    |   movel([0.251673, -1.221759, -2.667128, -0.823502, 1.570796, 1.822469],accel_mss,speed_ms,0,blend_radius_m)
    |   movel([0.252256, -1.224586, -2.665710, -0.822093, 1.570796, 1.823052],accel_mss,speed_ms,0,blend_radius_m)
    |   movel([0.252313, -1.225370, -2.665315, -0.821704, 1.570796, 1.823110],accel_mss,speed_ms,0,blend_radius_m)
    |   movel([0.252119, -1.226392, -2.664799, -0.821198, 1.570796, 1.822915],accel_mss,speed_ms,0,blend_radius_m)
    |   movel([0.252114, -1.226648, -2.664669, -0.821071, 1.570796, 1.822911],accel_mss,speed_ms,0,blend_radius_m)
    |   movel([0.252664, -1.227115, -2.664433, -0.820840, 1.570796, 1.823460],accel_mss,speed_ms,0,blend_radius_m)
    |   movel([0.252892, -1.227914, -2.664028, -0.820447, 1.570796, 1.823688],accel_mss,speed_ms,0,blend_radius_m)
    |   movel([0.253520, -1.231694, -2.662103, -0.818592, 1.570796, 1.824316],accel_mss,speed_ms,0,blend_radius_m)
    |   movel([0.254096, -1.235374, -2.660213, -0.816803, 1.570796, 1.824892],accel_mss,speed_ms,0,blend_radius_m)
    |   movel([0.255273, -1.240979, -2.657303, -0.814107, 1.570796, 1.826070],accel_mss,speed_ms,0,blend_radius_m)
    |   movel([0.255921, -1.243115, -2.656184, -0.813089, 1.570796, 1.826717],accel_mss,speed_ms,0,blend_radius_m)
    |   movel([0.256893, -1.245588, -2.654883, -0.811918, 1.570796, 1.827689],accel_mss,speed_ms,0,blend_radius_m)
    |   movel([0.258056, -1.247911, -2.653653, -0.810825, 1.570796, 1.828852],accel_mss,speed_ms,0,blend_radius_m)
    |   movel([0.259299, -1.249832, -2.652632, -0.809925, 1.570796, 1.830095],accel_mss,speed_ms,0,blend_radius_m)
    |   movel([0.260770, -1.251552, -2.651713, -0.809124, 1.570796, 1.831566],accel_mss,speed_ms,0,blend_radius_m)
    |   movel([0.262149, -1.252766, -2.651063, -0.808560, 1.570796, 1.832945],accel_mss,speed_ms,0,blend_radius_m)
    |   movel([0.263720, -1.253774, -2.650522, -0.808094, 1.570796, 1.834516],accel_mss,speed_ms,0,blend_radius_m)
    |   movel([0.265017, -1.254154, -2.650317, -0.807918, 1.570796, 1.835813],accel_mss,speed_ms,0,blend_radius_m)
    |   movel([0.266576, -1.254061, -2.650367, -0.807961, 1.570796, 1.837372],accel_mss,speed_ms,0,blend_radius_m)
    |   movel([0.268162, -1.253521, -2.650657, -0.808210, 1.570796, 1.838958],accel_mss,speed_ms,0,blend_radius_m)
    |   movel([0.268641, -1.253267, -2.650794, -0.808328, 1.570796, 1.839437],accel_mss,speed_ms,0,blend_radius_m)
    |   movel([0.270173, -1.252133, -2.651402, -0.808854, 1.570796, 1.840969],accel_mss,speed_ms,0,blend_radius_m)
    |   movel([0.271779, -1.250504, -2.652273, -0.809612, 1.570796, 1.842575],accel_mss,speed_ms,0,blend_radius_m)
    |   movel([0.273303, -1.248559, -2.653309, -0.810521, 1.570796, 1.844100],accel_mss,speed_ms,0,blend_radius_m)
    |   movel([0.274592, -1.246469, -2.654417, -0.811503, 1.570796, 1.845389],accel_mss,speed_ms,0,blend_radius_m)
    |   movel([0.275448, -1.244543, -2.655434, -0.812412, 1.570796, 1.846245],accel_mss,speed_ms,0,blend_radius_m)
    |   movel([0.276254, -1.241932, -2.656805, -0.813652, 1.570796, 1.847050],accel_mss,speed_ms,0,blend_radius_m)
    |   movel([0.276891, -1.239150, -2.658257, -0.814983, 1.570796, 1.847687],accel_mss,speed_ms,0,blend_radius_m)
    |   movel([0.277227, -1.236646, -2.659556, -0.816187, 1.570796, 1.848023],accel_mss,speed_ms,0,blend_radius_m)
    |   movel([0.277345, -1.234191, -2.660822, -0.817376, 1.570796, 1.848141],accel_mss,speed_ms,0,blend_radius_m)
    |   movel([0.277297, -1.231803, -2.662047, -0.818539, 1.570796, 1.848093],accel_mss,speed_ms,0,blend_radius_m)
    |   movel([0.277086, -1.229560, -2.663192, -0.819637, 1.570796, 1.847882],accel_mss,speed_ms,0,blend_radius_m)
    |   movel([0.276698, -1.227409, -2.664285, -0.820696, 1.570796, 1.847494],accel_mss,speed_ms,0,blend_radius_m)
    |   movel([0.276147, -1.225413, -2.665293, -0.821683, 1.570796, 1.846943],accel_mss,speed_ms,0,blend_radius_m)
    |   movel([0.275424, -1.223525, -2.666243, -0.822621, 1.570796, 1.846220],accel_mss,speed_ms,0,blend_radius_m)
    |   movel([0.274540, -1.221803, -2.667106, -0.823480, 1.570796, 1.845336],accel_mss,speed_ms,0,blend_radius_m)
    |   movel([0.273482, -1.220215, -2.667899, -0.824275, 1.570796, 1.844278],accel_mss,speed_ms,0,blend_radius_m)
    |   movel([0.272482, -1.219065, -2.668471, -0.824852, 1.570796, 1.843279],accel_mss,speed_ms,0,blend_radius_m)
    |   movel([0.272133, -1.218838, -2.668584, -0.824967, 1.570796, 1.842930],accel_mss,speed_ms,0,blend_radius_m)
    |   movel([0.271831, -1.218816, -2.668595, -0.824978, 1.570796, 1.842627],accel_mss,speed_ms,0,blend_radius_m)
    |   movel([0.271376, -1.219063, -2.668473, -0.824854, 1.570796, 1.842172],accel_mss,speed_ms,0,blend_radius_m)
    |   movel([0.271187, -1.219431, -2.668289, -0.824668, 1.570796, 1.841984],accel_mss,speed_ms,0,blend_radius_m)
    |   movel([0.271361, -1.219988, -2.668012, -0.824389, 1.570796, 1.842158],accel_mss,speed_ms,0,blend_radius_m)
    |   movel([0.271964, -1.220817, -2.667599, -0.823973, 1.570796, 1.842761],accel_mss,speed_ms,0,blend_radius_m)
    |   movel([0.273182, -1.222548, -2.666734, -0.823108, 1.570796, 1.843978],accel_mss,speed_ms,0,blend_radius_m)
    |   movel([0.274184, -1.224447, -2.665780, -0.822162, 1.570796, 1.844980],accel_mss,speed_ms,0,blend_radius_m)
    |   movel([0.274992, -1.226530, -2.664729, -0.821130, 1.570796, 1.845788],accel_mss,speed_ms,0,blend_radius_m)
    |   movel([0.275580, -1.228751, -2.663604, -0.820035, 1.570796, 1.846376],accel_mss,speed_ms,0,blend_radius_m)
    |   movel([0.275960, -1.231114, -2.662400, -0.818876, 1.570796, 1.846756],accel_mss,speed_ms,0,blend_radius_m)
    |   movel([0.276124, -1.233583, -2.661135, -0.817671, 1.570796, 1.846920],accel_mss,speed_ms,0,blend_radius_m)
    |   movel([0.276071, -1.236144, -2.659815, -0.816430, 1.570796, 1.846867],accel_mss,speed_ms,0,blend_radius_m)
    |   movel([0.275805, -1.238781, -2.658448, -0.815159, 1.570796, 1.846602],accel_mss,speed_ms,0,blend_radius_m)
    |   movel([0.275419, -1.240897, -2.657346, -0.814146, 1.570796, 1.846215],accel_mss,speed_ms,0,blend_radius_m)
    |   movel([0.274837, -1.243056, -2.656215, -0.813117, 1.570796, 1.845633],accel_mss,speed_ms,0,blend_radius_m)
    |   movel([0.274120, -1.244995, -2.655195, -0.812198, 1.570796, 1.844916],accel_mss,speed_ms,0,blend_radius_m)
    |   movel([0.273176, -1.246938, -2.654169, -0.811282, 1.570796, 1.843972],accel_mss,speed_ms,0,blend_radius_m)
    |   movel([0.272189, -1.248540, -2.653319, -0.810530, 1.570796, 1.842985],accel_mss,speed_ms,0,blend_radius_m)
    |   movel([0.271011, -1.250081, -2.652499, -0.809809, 1.570796, 1.841807],accel_mss,speed_ms,0,blend_radius_m)
    |   movel([0.269852, -1.251241, -2.651879, -0.809268, 1.570796, 1.840649],accel_mss,speed_ms,0,blend_radius_m)
    |   movel([0.268535, -1.252186, -2.651374, -0.808829, 1.570796, 1.839332],accel_mss,speed_ms,0,blend_radius_m)
    |   movel([0.267582, -1.252648, -2.651126, -0.808615, 1.570796, 1.838378],accel_mss,speed_ms,0,blend_radius_m)
    |   movel([0.266683, -1.252879, -2.651002, -0.808507, 1.570796, 1.837480],accel_mss,speed_ms,0,blend_radius_m)
    |   movel([0.265766, -1.252881, -2.651001, -0.808507, 1.570796, 1.836563],accel_mss,speed_ms,0,blend_radius_m)
    |   movel([0.264751, -1.252662, -2.651119, -0.808608, 1.570796, 1.835547],accel_mss,speed_ms,0,blend_radius_m)
    |   movel([0.263859, -1.252274, -2.651327, -0.808788, 1.570796, 1.834655],accel_mss,speed_ms,0,blend_radius_m)
    |   movel([0.263122, -1.251705, -2.651631, -0.809052, 1.570796, 1.833919],accel_mss,speed_ms,0,blend_radius_m)
    |   movel([0.260735, -1.249084, -2.653030, -0.810275, 1.570796, 1.831531],accel_mss,speed_ms,0,blend_radius_m)
    |   movel([0.258421, -1.246199, -2.654560, -0.811630, 1.570796, 1.829217],accel_mss,speed_ms,0,blend_radius_m)
    |   movel([0.258350, -1.245788, -2.654777, -0.811824, 1.570796, 1.829146],accel_mss,speed_ms,0,blend_radius_m)
    |   movel([0.258596, -1.245287, -2.655042, -0.812060, 1.570796, 1.829392],accel_mss,speed_ms,0,blend_radius_m)
    |   movel([0.258596, -1.244631, -2.655387, -0.812370, 1.570796, 1.829393],accel_mss,speed_ms,0,blend_radius_m)
    |   movel([0.258518, -1.243848, -2.655800, -0.812742, 1.570796, 1.829314],accel_mss,speed_ms,0,blend_radius_m)
    |   movel([0.258893, -1.242963, -2.656264, -0.813162, 1.570796, 1.829689],accel_mss,speed_ms,0,blend_radius_m)
    |   movel([0.259695, -1.242085, -2.656725, -0.813579, 1.570796, 1.830491],accel_mss,speed_ms,0,blend_radius_m)
    |   movel([0.260821, -1.241329, -2.657120, -0.813940, 1.570796, 1.831618],accel_mss,speed_ms,0,blend_radius_m)
    |   movel([0.261962, -1.240850, -2.657371, -0.814169, 1.570796, 1.832758],accel_mss,speed_ms,0,blend_radius_m)
    |   movel([0.263259, -1.240549, -2.657527, -0.814312, 1.570796, 1.834056],accel_mss,speed_ms,0,blend_radius_m)
    |   movel([0.264431, -1.240462, -2.657573, -0.814354, 1.570796, 1.835227],accel_mss,speed_ms,0,blend_radius_m)
    |   movel([0.265143, -1.240658, -2.657471, -0.814260, 1.570796, 1.835939],accel_mss,speed_ms,0,blend_radius_m)
    |   movel([0.265362, -1.240773, -2.657411, -0.814205, 1.570796, 1.836158],accel_mss,speed_ms,0,blend_radius_m)
    |   movel([0.266050, -1.240887, -2.657351, -0.814151, 1.570796, 1.836847],accel_mss,speed_ms,0,blend_radius_m)
    |   movel([0.266350, -1.240866, -2.657362, -0.814161, 1.570796, 1.837146],accel_mss,speed_ms,0,blend_radius_m)
    |   movel([0.266402, -1.240980, -2.657303, -0.814107, 1.570796, 1.837198],accel_mss,speed_ms,0,blend_radius_m)
    |   movel([0.266237, -1.241186, -2.657195, -0.814008, 1.570796, 1.837033],accel_mss,speed_ms,0,blend_radius_m)
    |   movel([0.265247, -1.241887, -2.656828, -0.813674, 1.570796, 1.836043],accel_mss,speed_ms,0,blend_radius_m)
    |   movel([0.264579, -1.242566, -2.656473, -0.813351, 1.570796, 1.835376],accel_mss,speed_ms,0,blend_radius_m)
    |   movel([0.263427, -1.244142, -2.655645, -0.812602, 1.570796, 1.834224],accel_mss,speed_ms,0,blend_radius_m)
    |   movel([0.262984, -1.245097, -2.655142, -0.812150, 1.570796, 1.833780],accel_mss,speed_ms,0,blend_radius_m)
    |   movel([0.262406, -1.247398, -2.653925, -0.811066, 1.570796, 1.833203],accel_mss,speed_ms,0,blend_radius_m)
    |   movel([0.262377, -1.248322, -2.653435, -0.810632, 1.570796, 1.833173],accel_mss,speed_ms,0,blend_radius_m)
    |   movel([0.262798, -1.250016, -2.652534, -0.809839, 1.570796, 1.833595],accel_mss,speed_ms,0,blend_radius_m)
    |   movel([0.263763, -1.251456, -2.651764, -0.809168, 1.570796, 1.834559],accel_mss,speed_ms,0,blend_radius_m)
    |   movel([0.264797, -1.252084, -2.651429, -0.808877, 1.570796, 1.835593],accel_mss,speed_ms,0,blend_radius_m)
    |   movel([0.265194, -1.252000, -2.651474, -0.808915, 1.570796, 1.835990],accel_mss,speed_ms,0,blend_radius_m)
    |   movel([0.265517, -1.251643, -2.651665, -0.809082, 1.570796, 1.836314],accel_mss,speed_ms,0,blend_radius_m)
    |   movel([0.265537, -1.251456, -2.651764, -0.809168, 1.570796, 1.836334],accel_mss,speed_ms,0,blend_radius_m)
    |   movel([0.264819, -1.250247, -2.652411, -0.809732, 1.570796, 1.835616],accel_mss,speed_ms,0,blend_radius_m)
    |   movel([0.264102, -1.249179, -2.652979, -0.810230, 1.570796, 1.834899],accel_mss,speed_ms,0,blend_radius_m)
    |   movel([0.263717, -1.248165, -2.653518, -0.810705, 1.570796, 1.834513],accel_mss,speed_ms,0,blend_radius_m)
    |   movel([0.263635, -1.247105, -2.654081, -0.811204, 1.570796, 1.834431],accel_mss,speed_ms,0,blend_radius_m)
    |   movel([0.263836, -1.245902, -2.654717, -0.811770, 1.570796, 1.834632],accel_mss,speed_ms,0,blend_radius_m)
    |   movel([0.264366, -1.244503, -2.655455, -0.812431, 1.570796, 1.835162],accel_mss,speed_ms,0,blend_radius_m)
    |   movel([0.265141, -1.243328, -2.656073, -0.812988, 1.570796, 1.835937],accel_mss,speed_ms,0,blend_radius_m)
    |   movel([0.266125, -1.242431, -2.656543, -0.813414, 1.570796, 1.836921],accel_mss,speed_ms,0,blend_radius_m)
    |   movel([0.267647, -1.241694, -2.656929, -0.813766, 1.570796, 1.838444],accel_mss,speed_ms,0,blend_radius_m)
    |   movel([0.268011, -1.241513, -2.657024, -0.813852, 1.570796, 1.838807],accel_mss,speed_ms,0,blend_radius_m)
    |   movel([0.268485, -1.241158, -2.657209, -0.814021, 1.570796, 1.839281],accel_mss,speed_ms,0,blend_radius_m)
    |   movel([0.268713, -1.241026, -2.657278, -0.814084, 1.570796, 1.839509],accel_mss,speed_ms,0,blend_radius_m)
    |   movel([0.268748, -1.241410, -2.657078, -0.813901, 1.570796, 1.839544],accel_mss,speed_ms,0,blend_radius_m)
    |   movel([0.269472, -1.242542, -2.656485, -0.813362, 1.570796, 1.840268],accel_mss,speed_ms,0,blend_radius_m)
    |   movel([0.270218, -1.243593, -2.655933, -0.812862, 1.570796, 1.841015],accel_mss,speed_ms,0,blend_radius_m)
    |   movel([0.270715, -1.244043, -2.655697, -0.812649, 1.570796, 1.841511],accel_mss,speed_ms,0,blend_radius_m)
    |   movel([0.271107, -1.244195, -2.655617, -0.812577, 1.570796, 1.841903],accel_mss,speed_ms,0,blend_radius_m)
    |   movel([0.271501, -1.244167, -2.655632, -0.812590, 1.570796, 1.842297],accel_mss,speed_ms,0,blend_radius_m)
    |   movel([0.271816, -1.243974, -2.655733, -0.812682, 1.570796, 1.842613],accel_mss,speed_ms,0,blend_radius_m)
    |   movel([0.272009, -1.243666, -2.655895, -0.812828, 1.570796, 1.842805],accel_mss,speed_ms,0,blend_radius_m)
    |   movel([0.272002, -1.243499, -2.655983, -0.812907, 1.570796, 1.842799],accel_mss,speed_ms,0,blend_radius_m)
    |   movel([0.270423, -1.241210, -2.657183, -0.813997, 1.570796, 1.841220],accel_mss,speed_ms,0,blend_radius_m)
    |   movel([0.269852, -1.240023, -2.657802, -0.814564, 1.570796, 1.840649],accel_mss,speed_ms,0,blend_radius_m)
    |   movel([0.269473, -1.238726, -2.658477, -0.815186, 1.570796, 1.840269],accel_mss,speed_ms,0,blend_radius_m)
    |   movel([0.269282, -1.237334, -2.659200, -0.815856, 1.570796, 1.840079],accel_mss,speed_ms,0,blend_radius_m)
    |   movel([0.269385, -1.234643, -2.660589, -0.817156, 1.570796, 1.840181],accel_mss,speed_ms,0,blend_radius_m)
    |   movel([0.269553, -1.233087, -2.661389, -0.817912, 1.570796, 1.840349],accel_mss,speed_ms,0,blend_radius_m)
    |   movel([0.269726, -1.232780, -2.661547, -0.818062, 1.570796, 1.840522],accel_mss,speed_ms,0,blend_radius_m)
    |   movel([0.271064, -1.233074, -2.661396, -0.817919, 1.570796, 1.841860],accel_mss,speed_ms,0,blend_radius_m)
    |   movel([0.272118, -1.233330, -2.661265, -0.817794, 1.570796, 1.842915],accel_mss,speed_ms,0,blend_radius_m)
    |   movel([0.274209, -1.233442, -2.661207, -0.817740, 1.570796, 1.845005],accel_mss,speed_ms,0,blend_radius_m)
    |   movel([0.274650, -1.233227, -2.661317, -0.817844, 1.570796, 1.845446],accel_mss,speed_ms,0,blend_radius_m)
    |   movel([0.274831, -1.232962, -2.661453, -0.817973, 1.570796, 1.845627],accel_mss,speed_ms,0,blend_radius_m)
    |   movel([0.274895, -1.232796, -2.661539, -0.818054, 1.570796, 1.845691],accel_mss,speed_ms,0,blend_radius_m)
    |   movel([0.274868, -1.232472, -2.661705, -0.818212, 1.570796, 1.845664],accel_mss,speed_ms,0,blend_radius_m)
    |   movel([0.274650, -1.232351, -2.661767, -0.818271, 1.570796, 1.845446],accel_mss,speed_ms,0,blend_radius_m)
    |   movel([0.273622, -1.232213, -2.661838, -0.818339, 1.570796, 1.844418],accel_mss,speed_ms,0,blend_radius_m)
    |   movel([0.272503, -1.232068, -2.661912, -0.818409, 1.570796, 1.843299],accel_mss,speed_ms,0,blend_radius_m)
    |   movel([0.271457, -1.231749, -2.662075, -0.818565, 1.570796, 1.842253],accel_mss,speed_ms,0,blend_radius_m)
    |   movel([0.270643, -1.231335, -2.662286, -0.818767, 1.570796, 1.841439],accel_mss,speed_ms,0,blend_radius_m)
    |   movel([0.270352, -1.230900, -2.662509, -0.818980, 1.570796, 1.841148],accel_mss,speed_ms,0,blend_radius_m)
    |   movel([0.270297, -1.230746, -2.662588, -0.819056, 1.570796, 1.841094],accel_mss,speed_ms,0,blend_radius_m)
    |   movel([0.269838, -1.230421, -2.662753, -0.819214, 1.570796, 1.840634],accel_mss,speed_ms,0,blend_radius_m)
    |   movel([0.269735, -1.230051, -2.662942, -0.819396, 1.570796, 1.840531],accel_mss,speed_ms,0,blend_radius_m)
    |   movel([0.269575, -1.227075, -2.664454, -0.820861, 1.570796, 1.840372],accel_mss,speed_ms,0,blend_radius_m)
    |   movel([0.269978, -1.227005, -2.664489, -0.820895, 1.570796, 1.840774],accel_mss,speed_ms,0,blend_radius_m)
    |   movel([0.270364, -1.227000, -2.664491, -0.820897, 1.570796, 1.841160],accel_mss,speed_ms,0,blend_radius_m)
    |   movel([0.272607, -1.226884, -2.664550, -0.820955, 1.570796, 1.843404],accel_mss,speed_ms,0,blend_radius_m)
    |   movel([0.273200, -1.226702, -2.664642, -0.821045, 1.570796, 1.843996],accel_mss,speed_ms,0,blend_radius_m)
    |   movel([0.273592, -1.226427, -2.664781, -0.821181, 1.570796, 1.844388],accel_mss,speed_ms,0,blend_radius_m)
    |   movel([0.273858, -1.226019, -2.664987, -0.821382, 1.570796, 1.844654],accel_mss,speed_ms,0,blend_radius_m)
    |   movel([0.273809, -1.225748, -2.665124, -0.821517, 1.570796, 1.844605],accel_mss,speed_ms,0,blend_radius_m)
    |   movel([0.273385, -1.225635, -2.665181, -0.821573, 1.570796, 1.844181],accel_mss,speed_ms,0,blend_radius_m)
    |   movel([0.272519, -1.225697, -2.665150, -0.821542, 1.570796, 1.843315],accel_mss,speed_ms,0,blend_radius_m)
    |   movel([0.271938, -1.225740, -2.665128, -0.821521, 1.570796, 1.842734],accel_mss,speed_ms,0,blend_radius_m)
    |   movel([0.270210, -1.225590, -2.665204, -0.821595, 1.570796, 1.841006],accel_mss,speed_ms,0,blend_radius_m)
    |   movel([0.269603, -1.225372, -2.665314, -0.821703, 1.570796, 1.840399],accel_mss,speed_ms,0,blend_radius_m)
    |   movel([0.269293, -1.225101, -2.665450, -0.821837, 1.570796, 1.840089],accel_mss,speed_ms,0,blend_radius_m)
    |   movel([0.269082, -1.224608, -2.665699, -0.822082, 1.570796, 1.839879],accel_mss,speed_ms,0,blend_radius_m)
    |   movel([0.268295, -1.220623, -2.667696, -0.824070, 1.570796, 1.839091],accel_mss,speed_ms,0,blend_radius_m)
    |   movel([0.268094, -1.218191, -2.668905, -0.825293, 1.570796, 1.838890],accel_mss,speed_ms,0,blend_radius_m)
    |   movel([0.268165, -1.215682, -2.670146, -0.826561, 1.570796, 1.838962],accel_mss,speed_ms,0,blend_radius_m)
    |   movel([0.268510, -1.212727, -2.671599, -0.828063, 1.570796, 1.839307],accel_mss,speed_ms,0,blend_radius_m)
    |   movel([0.269312, -1.208863, -2.673483, -0.830043, 1.570796, 1.840109],accel_mss,speed_ms,0,blend_radius_m)
    |   movel([0.270551, -1.205077, -2.675313, -0.831998, 1.570796, 1.841347],accel_mss,speed_ms,0,blend_radius_m)
    |   movel([0.272166, -1.201531, -2.677013, -0.833845, 1.570796, 1.842962],accel_mss,speed_ms,0,blend_radius_m)
    |   movel([0.273066, -1.199947, -2.677768, -0.834674, 1.570796, 1.843863],accel_mss,speed_ms,0,blend_radius_m)
    |   movel([0.274103, -1.198381, -2.678512, -0.835497, 1.570796, 1.844900],accel_mss,speed_ms,0,blend_radius_m)
    |   movel([0.275647, -1.196414, -2.679442, -0.836533, 1.570796, 1.846443],accel_mss,speed_ms,0,blend_radius_m)
    |   movel([0.277625, -1.194250, -2.680460, -0.837679, 1.570796, 1.848421],accel_mss,speed_ms,0,blend_radius_m)
    |   movel([0.279732, -1.192197, -2.681422, -0.838771, 1.570796, 1.850529],accel_mss,speed_ms,0,blend_radius_m)
    |   movel([0.281670, -1.190580, -2.682175, -0.839633, 1.570796, 1.852466],accel_mss,speed_ms,0,blend_radius_m)
    |   movel([0.283687, -1.189141, -2.682844, -0.840404, 1.570796, 1.854484],accel_mss,speed_ms,0,blend_radius_m)
    |   movel([0.285751, -1.187861, -2.683437, -0.841091, 1.570796, 1.856547],accel_mss,speed_ms,0,blend_radius_m)
    |   movel([0.287875, -1.186725, -2.683962, -0.841702, 1.570796, 1.858671],accel_mss,speed_ms,0,blend_radius_m)
    |   movel([0.290006, -1.185763, -2.684405, -0.842221, 1.570796, 1.860802],accel_mss,speed_ms,0,blend_radius_m)
    |   movel([0.292162, -1.184969, -2.684770, -0.842650, 1.570796, 1.862959],accel_mss,speed_ms,0,blend_radius_m)
    |   movel([0.294283, -1.184372, -2.685044, -0.842973, 1.570796, 1.865079],accel_mss,speed_ms,0,blend_radius_m)
    |   movel([0.296396, -1.183955, -2.685235, -0.843198, 1.570796, 1.867192],accel_mss,speed_ms,0,blend_radius_m)
    |   movel([0.298436, -1.183735, -2.685336, -0.843318, 1.570796, 1.869233],accel_mss,speed_ms,0,blend_radius_m)
    |   movel([0.301164, -1.183724, -2.685341, -0.843324, 1.570796, 1.871961],accel_mss,speed_ms,0,blend_radius_m)
    |   movel([0.303716, -1.184044, -2.685195, -0.843150, 1.570796, 1.874512],accel_mss,speed_ms,0,blend_radius_m)
    |   movel([0.305964, -1.184677, -2.684904, -0.842808, 1.570796, 1.876761],accel_mss,speed_ms,0,blend_radius_m)
    |   movel([0.307966, -1.185647, -2.684459, -0.842284, 1.570796, 1.878762],accel_mss,speed_ms,0,blend_radius_m)
    |   movel([0.309607, -1.186887, -2.683887, -0.841615, 1.570796, 1.880403],accel_mss,speed_ms,0,blend_radius_m)
    |   movel([0.310946, -1.188428, -2.683175, -0.840786, 1.570796, 1.881742],accel_mss,speed_ms,0,blend_radius_m)
    |   movel([0.311905, -1.190185, -2.682359, -0.839844, 1.570796, 1.882701],accel_mss,speed_ms,0,blend_radius_m)
    |   movel([0.312501, -1.192206, -2.681417, -0.838766, 1.570796, 1.883297],accel_mss,speed_ms,0,blend_radius_m)
    |   movel([0.312796, -1.195034, -2.680092, -0.837263, 1.570796, 1.883592],accel_mss,speed_ms,0,blend_radius_m)
    |   movel([0.312643, -1.198070, -2.678659, -0.835660, 1.570796, 1.883439],accel_mss,speed_ms,0,blend_radius_m)
    |   movel([0.312002, -1.202419, -2.676589, -0.833381, 1.570796, 1.882798],accel_mss,speed_ms,0,blend_radius_m)
    |   movel([0.311133, -1.206813, -2.674476, -0.831100, 1.570796, 1.881929],accel_mss,speed_ms,0,blend_radius_m)
    |   movel([0.309766, -1.212476, -2.671722, -0.828191, 1.570796, 1.880562],accel_mss,speed_ms,0,blend_radius_m)
    |   movel([0.308178, -1.218145, -2.668928, -0.825316, 1.570796, 1.878974],accel_mss,speed_ms,0,blend_radius_m)
    |   movel([0.305985, -1.225255, -2.665373, -0.821761, 1.570796, 1.876782],accel_mss,speed_ms,0,blend_radius_m)
    |   movel([0.296721, -1.253611, -2.650609, -0.808169, 1.570796, 1.867517],accel_mss,speed_ms,0,blend_radius_m)
    |   movel([0.294612, -1.260515, -2.646870, -0.805004, 1.570796, 1.865408],accel_mss,speed_ms,0,blend_radius_m)
    |   movel([0.292702, -1.267312, -2.643132, -0.801946, 1.570796, 1.863498],accel_mss,speed_ms,0,blend_radius_m)
    |   movel([0.291421, -1.272421, -2.640284, -0.799684, 1.570796, 1.862217],accel_mss,speed_ms,0,blend_radius_m)
    |   movel([0.290344, -1.277443, -2.637454, -0.797492, 1.570796, 1.861140],accel_mss,speed_ms,0,blend_radius_m)
    |   movel([0.289565, -1.281959, -2.634881, -0.795548, 1.570796, 1.860362],accel_mss,speed_ms,0,blend_radius_m)
    |   movel([0.289021, -1.286374, -2.632342, -0.793673, 1.570796, 1.859818],accel_mss,speed_ms,0,blend_radius_m)
    |   movel([0.288720, -1.290024, -2.630224, -0.792141, 1.570796, 1.859516],accel_mss,speed_ms,0,blend_radius_m)
    |   movel([0.288628, -1.292746, -2.628633, -0.791010, 1.570796, 1.859425],accel_mss,speed_ms,0,blend_radius_m)
    |   movel([0.288730, -1.294853, -2.627395, -0.790140, 1.570796, 1.859526],accel_mss,speed_ms,0,blend_radius_m)
    |   movel([0.289030, -1.296545, -2.626397, -0.789446, 1.570796, 1.859827],accel_mss,speed_ms,0,blend_radius_m)
    |   movel([0.289400, -1.297463, -2.625854, -0.789071, 1.570796, 1.860196],accel_mss,speed_ms,0,blend_radius_m)
    |   movel([0.290019, -1.298360, -2.625322, -0.788706, 1.570796, 1.860816],accel_mss,speed_ms,0,blend_radius_m)
    |   movel([0.290702, -1.299067, -2.624903, -0.788419, 1.570796, 1.861498],accel_mss,speed_ms,0,blend_radius_m)
    |   movel([0.291185, -1.299131, -2.624865, -0.788393, 1.570796, 1.861982],accel_mss,speed_ms,0,blend_radius_m)
    |   movel([0.291568, -1.298901, -2.625002, -0.788487, 1.570796, 1.862364],accel_mss,speed_ms,0,blend_radius_m)
    |   movel([0.291720, -1.298581, -2.625192, -0.788616, 1.570796, 1.862516],accel_mss,speed_ms,0,blend_radius_m)
    |   movel([0.291581, -1.298122, -2.625464, -0.788803, 1.570796, 1.862378],accel_mss,speed_ms,0,blend_radius_m)
    |   movel([0.290575, -1.296692, -2.626310, -0.789386, 1.570796, 1.861371],accel_mss,speed_ms,0,blend_radius_m)
    |   movel([0.290158, -1.295653, -2.626924, -0.789812, 1.570796, 1.860954],accel_mss,speed_ms,0,blend_radius_m)
    |   movel([0.289893, -1.294509, -2.627598, -0.790282, 1.570796, 1.860689],accel_mss,speed_ms,0,blend_radius_m)
    |   movel([0.289830, -1.293400, -2.628250, -0.790739, 1.570796, 1.860626],accel_mss,speed_ms,0,blend_radius_m)
    |   movel([0.289909, -1.292862, -2.628565, -0.790962, 1.570796, 1.860705],accel_mss,speed_ms,0,blend_radius_m)
    |   movel([0.290523, -1.292619, -2.628708, -0.791062, 1.570796, 1.861320],accel_mss,speed_ms,0,blend_radius_m)
    |   movel([0.290785, -1.292414, -2.628828, -0.791147, 1.570796, 1.861581],accel_mss,speed_ms,0,blend_radius_m)
    |   movel([0.291653, -1.291164, -2.629559, -0.791666, 1.570796, 1.862449],accel_mss,speed_ms,0,blend_radius_m)
    |   movel([0.292323, -1.290260, -2.630086, -0.792042, 1.570796, 1.863119],accel_mss,speed_ms,0,blend_radius_m)
    |   movel([0.293176, -1.289368, -2.630606, -0.792415, 1.570796, 1.863972],accel_mss,speed_ms,0,blend_radius_m)
    |   movel([0.294123, -1.288573, -2.631068, -0.792748, 1.570796, 1.864920],accel_mss,speed_ms,0,blend_radius_m)
    |   movel([0.295077, -1.287958, -2.631425, -0.793006, 1.570796, 1.865873],accel_mss,speed_ms,0,blend_radius_m)
    |   movel([0.296104, -1.287510, -2.631685, -0.793194, 1.570796, 1.866900],accel_mss,speed_ms,0,blend_radius_m)
    |   movel([0.297277, -1.287210, -2.631858, -0.793320, 1.570796, 1.868073],accel_mss,speed_ms,0,blend_radius_m)
    |   movel([0.298394, -1.287097, -2.631924, -0.793368, 1.570796, 1.869190],accel_mss,speed_ms,0,blend_radius_m)
    |   movel([0.299744, -1.287306, -2.631803, -0.793280, 1.570796, 1.870541],accel_mss,speed_ms,0,blend_radius_m)
    |   movel([0.300143, -1.287250, -2.631835, -0.793304, 1.570796, 1.870939],accel_mss,speed_ms,0,blend_radius_m)
    |   movel([0.300433, -1.287053, -2.631949, -0.793386, 1.570796, 1.871229],accel_mss,speed_ms,0,blend_radius_m)
    |   movel([0.300623, -1.286735, -2.632134, -0.793521, 1.570796, 1.871420],accel_mss,speed_ms,0,blend_radius_m)
    |   movel([0.300638, -1.286513, -2.632262, -0.793614, 1.570796, 1.871434],accel_mss,speed_ms,0,blend_radius_m)
    |   movel([0.300532, -1.286361, -2.632349, -0.793678, 1.570796, 1.871329],accel_mss,speed_ms,0,blend_radius_m)
    |   movel([0.299923, -1.286102, -2.632499, -0.793788, 1.570796, 1.870720],accel_mss,speed_ms,0,blend_radius_m)
    |   movel([0.299003, -1.285987, -2.632566, -0.793836, 1.570796, 1.869799],accel_mss,speed_ms,0,blend_radius_m)
    |   movel([0.296600, -1.286246, -2.632416, -0.793727, 1.570796, 1.867396],accel_mss,speed_ms,0,blend_radius_m)
    |   movel([0.297155, -1.285652, -2.632759, -0.793978, 1.570796, 1.867951],accel_mss,speed_ms,0,blend_radius_m)
    |   movel([0.298363, -1.284645, -2.633340, -0.794404, 1.570796, 1.869159],accel_mss,speed_ms,0,blend_radius_m)
    |   movel([0.300011, -1.283745, -2.633857, -0.794787, 1.570796, 1.870807],accel_mss,speed_ms,0,blend_radius_m)
    |   movel([0.301709, -1.283124, -2.634214, -0.795051, 1.570796, 1.872505],accel_mss,speed_ms,0,blend_radius_m)
    |   movel([0.302405, -1.282985, -2.634294, -0.795110, 1.570796, 1.873201],accel_mss,speed_ms,0,blend_radius_m)
    |   movel([0.303656, -1.282958, -2.634309, -0.795122, 1.570796, 1.874452],accel_mss,speed_ms,0,blend_radius_m)
    |   movel([0.304101, -1.282840, -2.634377, -0.795172, 1.570796, 1.874898],accel_mss,speed_ms,0,blend_radius_m)
    |   movel([0.304410, -1.282615, -2.634506, -0.795268, 1.570796, 1.875206],accel_mss,speed_ms,0,blend_radius_m)
    |   movel([0.304606, -1.282291, -2.634692, -0.795407, 1.570796, 1.875402],accel_mss,speed_ms,0,blend_radius_m)
    |   movel([0.304597, -1.281997, -2.634860, -0.795532, 1.570796, 1.875394],accel_mss,speed_ms,0,blend_radius_m)
    |   movel([0.304377, -1.281859, -2.634939, -0.795591, 1.570796, 1.875173],accel_mss,speed_ms,0,blend_radius_m)
    |   movel([0.303093, -1.281851, -2.634943, -0.795595, 1.570796, 1.873889],accel_mss,speed_ms,0,blend_radius_m)
    |   movel([0.301425, -1.282160, -2.634766, -0.795462, 1.570796, 1.872221],accel_mss,speed_ms,0,blend_radius_m)
    |   movel([0.299834, -1.282753, -2.634427, -0.795209, 1.570796, 1.870631],accel_mss,speed_ms,0,blend_radius_m)
    |   movel([0.298673, -1.283406, -2.634052, -0.794931, 1.570796, 1.869470],accel_mss,speed_ms,0,blend_radius_m)
    |   movel([0.297438, -1.284299, -2.633539, -0.794551, 1.570796, 1.868235],accel_mss,speed_ms,0,blend_radius_m)
    |   movel([0.296316, -1.285278, -2.632975, -0.794136, 1.570796, 1.867112],accel_mss,speed_ms,0,blend_radius_m)
    |   movel([0.295504, -1.286195, -2.632445, -0.793748, 1.570796, 1.866300],accel_mss,speed_ms,0,blend_radius_m)
    |   movel([0.295210, -1.286554, -2.632238, -0.793597, 1.570796, 1.866007],accel_mss,speed_ms,0,blend_radius_m)
    |   movel([0.294269, -1.287405, -2.631745, -0.793238, 1.570796, 1.865066],accel_mss,speed_ms,0,blend_radius_m)
    |   movel([0.293340, -1.288068, -2.631361, -0.792960, 1.570796, 1.864136],accel_mss,speed_ms,0,blend_radius_m)
    |   movel([0.292264, -1.289066, -2.630781, -0.792541, 1.570796, 1.863060],accel_mss,speed_ms,0,blend_radius_m)
    |   movel([0.291254, -1.290177, -2.630135, -0.792077, 1.570796, 1.862050],accel_mss,speed_ms,0,blend_radius_m)
    |   movel([0.290529, -1.291187, -2.629546, -0.791657, 1.570796, 1.861325],accel_mss,speed_ms,0,blend_radius_m)
    |   movel([0.289778, -1.292409, -2.628831, -0.791149, 1.570796, 1.860575],accel_mss,speed_ms,0,blend_radius_m)
    |   movel([0.289957, -1.289396, -2.630590, -0.792403, 1.570796, 1.860754],accel_mss,speed_ms,0,blend_radius_m)
    |   movel([0.290249, -1.285698, -2.632733, -0.793959, 1.570796, 1.861045],accel_mss,speed_ms,0,blend_radius_m)
    |   movel([0.290680, -1.282109, -2.634796, -0.795484, 1.570796, 1.861477],accel_mss,speed_ms,0,blend_radius_m)
    |   movel([0.291289, -1.278366, -2.636930, -0.797093, 1.570796, 1.862085],accel_mss,speed_ms,0,blend_radius_m)
    |   movel([0.292758, -1.271276, -2.640925, -0.800188, 1.570796, 1.863554],accel_mss,speed_ms,0,blend_radius_m)
    |   movel([0.293046, -1.270340, -2.641448, -0.800601, 1.570796, 1.863842],accel_mss,speed_ms,0,blend_radius_m)
    |   movel([0.293399, -1.269829, -2.641733, -0.800827, 1.570796, 1.864195],accel_mss,speed_ms,0,blend_radius_m)
    |   movel([0.293969, -1.269434, -2.641953, -0.801002, 1.570796, 1.864765],accel_mss,speed_ms,0,blend_radius_m)
    |   movel([0.294435, -1.269241, -2.642060, -0.801088, 1.570796, 1.865231],accel_mss,speed_ms,0,blend_radius_m)
    |   movel([0.294760, -1.269176, -2.642096, -0.801117, 1.570796, 1.865556],accel_mss,speed_ms,0,blend_radius_m)
    |   movel([0.295611, -1.269389, -2.641978, -0.801022, 1.570796, 1.866407],accel_mss,speed_ms,0,blend_radius_m)
    |   movel([0.296405, -1.269792, -2.641753, -0.800844, 1.570796, 1.867201],accel_mss,speed_ms,0,blend_radius_m)
    |   movel([0.297145, -1.270383, -2.641424, -0.800582, 1.570796, 1.867941],accel_mss,speed_ms,0,blend_radius_m)
    |   movel([0.297727, -1.271069, -2.641041, -0.800279, 1.570796, 1.868523],accel_mss,speed_ms,0,blend_radius_m)
    |   movel([0.298041, -1.271742, -2.640664, -0.799982, 1.570796, 1.868837],accel_mss,speed_ms,0,blend_radius_m)
    |   movel([0.298230, -1.272433, -2.640277, -0.799679, 1.570796, 1.869026],accel_mss,speed_ms,0,blend_radius_m)
    |   movel([0.301663, -1.271908, -2.640571, -0.799909, 1.570796, 1.872459],accel_mss,speed_ms,0,blend_radius_m)
    |   movel([0.302358, -1.271869, -2.640593, -0.799927, 1.570796, 1.873155],accel_mss,speed_ms,0,blend_radius_m)
    |   movel([0.303603, -1.272149, -2.640436, -0.799803, 1.570796, 1.874399],accel_mss,speed_ms,0,blend_radius_m)
    |   movel([0.304507, -1.272607, -2.640180, -0.799602, 1.570796, 1.875304],accel_mss,speed_ms,0,blend_radius_m)
    |   movel([0.305245, -1.273260, -2.639813, -0.799315, 1.570796, 1.876041],accel_mss,speed_ms,0,blend_radius_m)
    |   movel([0.305796, -1.274093, -2.639345, -0.798951, 1.570796, 1.876593],accel_mss,speed_ms,0,blend_radius_m)
    |   movel([0.306270, -1.275494, -2.638556, -0.798339, 1.570796, 1.877066],accel_mss,speed_ms,0,blend_radius_m)
    |   movel([0.306412, -1.275831, -2.638366, -0.798192, 1.570796, 1.877209],accel_mss,speed_ms,0,blend_radius_m)
    |   movel([0.306668, -1.276119, -2.638203, -0.798067, 1.570796, 1.877464],accel_mss,speed_ms,0,blend_radius_m)
    |   movel([0.307047, -1.275960, -2.638293, -0.798136, 1.570796, 1.877844],accel_mss,speed_ms,0,blend_radius_m)
    |   movel([0.307298, -1.275670, -2.638457, -0.798262, 1.570796, 1.878095],accel_mss,speed_ms,0,blend_radius_m)
    |   movel([0.307403, -1.275216, -2.638713, -0.798460, 1.570796, 1.878200],accel_mss,speed_ms,0,blend_radius_m)
    |   movel([0.307351, -1.274575, -2.639074, -0.798740, 1.570796, 1.878148],accel_mss,speed_ms,0,blend_radius_m)
    |   movel([0.307181, -1.273923, -2.639441, -0.799025, 1.570796, 1.877977],accel_mss,speed_ms,0,blend_radius_m)
    |   speed_ms = 0.005
    |   movel([0.307181, -1.264567, -2.634963, -0.812858, 1.570796, 1.877977],accel_mss,speed_ms,0,blend_radius_m)
    |   speed_ms = 0.040
    |   movel([0.304112, -1.269554, -2.632181, -0.810654, 1.570796, 1.874909],accel_mss,speed_ms,0,blend_radius_m)
    |   speed_ms = 0.005
    |   movel([0.304112, -1.278884, -2.636636, -0.796869, 1.570796, 1.874909],accel_mss,speed_ms,0,blend_radius_m)
    |   speed_ms = 0.025
    |   movel([0.304270, -1.278746, -2.636714, -0.796929, 1.570796, 1.875066],accel_mss,speed_ms,0,blend_radius_m)
    |   movel([0.304601, -1.278282, -2.636978, -0.797129, 1.570796, 1.875398],accel_mss,speed_ms,0,blend_radius_m)
    |   movel([0.304563, -1.277853, -2.637222, -0.797315, 1.570796, 1.875360],accel_mss,speed_ms,0,blend_radius_m)
    |   movel([0.303997, -1.277210, -2.637586, -0.797593, 1.570796, 1.874794],accel_mss,speed_ms,0,blend_radius_m)
    |   movel([0.303308, -1.276645, -2.637906, -0.797838, 1.570796, 1.874104],accel_mss,speed_ms,0,blend_radius_m)
    |   movel([0.302686, -1.276414, -2.638036, -0.797939, 1.570796, 1.873483],accel_mss,speed_ms,0,blend_radius_m)
    |   movel([0.301769, -1.276358, -2.638068, -0.797963, 1.570796, 1.872565],accel_mss,speed_ms,0,blend_radius_m)
    |   movel([0.300985, -1.276506, -2.637984, -0.797899, 1.570796, 1.871782],accel_mss,speed_ms,0,blend_radius_m)
    |   movel([0.300206, -1.276888, -2.637768, -0.797733, 1.570796, 1.871002],accel_mss,speed_ms,0,blend_radius_m)
    |   movel([0.298672, -1.278078, -2.637094, -0.797217, 1.570796, 1.869468],accel_mss,speed_ms,0,blend_radius_m)
    |   movel([0.297788, -1.277736, -2.637288, -0.797365, 1.570796, 1.868584],accel_mss,speed_ms,0,blend_radius_m)
    |   movel([0.296471, -1.277488, -2.637429, -0.797473, 1.570796, 1.867267],accel_mss,speed_ms,0,blend_radius_m)
    |   movel([0.294936, -1.277638, -2.637343, -0.797408, 1.570796, 1.865733],accel_mss,speed_ms,0,blend_radius_m)
    |   movel([0.293429, -1.278152, -2.637052, -0.797186, 1.570796, 1.864225],accel_mss,speed_ms,0,blend_radius_m)
    |   movel([0.292793, -1.278503, -2.636852, -0.797034, 1.570796, 1.863590],accel_mss,speed_ms,0,blend_radius_m)
    |   movel([0.292196, -1.278959, -2.636593, -0.796837, 1.570796, 1.862992],accel_mss,speed_ms,0,blend_radius_m)
    |   movel([0.291689, -1.279491, -2.636290, -0.796607, 1.570796, 1.862485],accel_mss,speed_ms,0,blend_radius_m)
    |   movel([0.291352, -1.280042, -2.635976, -0.796370, 1.570796, 1.862148],accel_mss,speed_ms,0,blend_radius_m)
    |   movel([0.291218, -1.280560, -2.635681, -0.796148, 1.570796, 1.862015],accel_mss,speed_ms,0,blend_radius_m)
    |   movel([0.291295, -1.280989, -2.635436, -0.795964, 1.570796, 1.862091],accel_mss,speed_ms,0,blend_radius_m)
    |   movel([0.291522, -1.281180, -2.635327, -0.795882, 1.570796, 1.862318],accel_mss,speed_ms,0,blend_radius_m)
    |   movel([0.291828, -1.281115, -2.635364, -0.795910, 1.570796, 1.862624],accel_mss,speed_ms,0,blend_radius_m)
    |   movel([0.292137, -1.280798, -2.635545, -0.796046, 1.570796, 1.862933],accel_mss,speed_ms,0,blend_radius_m)
    |   movel([0.292502, -1.279941, -2.636034, -0.796414, 1.570796, 1.863298],accel_mss,speed_ms,0,blend_radius_m)
    |   movel([0.292668, -1.279695, -2.636174, -0.796520, 1.570796, 1.863464],accel_mss,speed_ms,0,blend_radius_m)
    |   movel([0.293368, -1.279216, -2.636447, -0.796726, 1.570796, 1.864164],accel_mss,speed_ms,0,blend_radius_m)
    |   movel([0.294384, -1.278800, -2.636683, -0.796905, 1.570796, 1.865181],accel_mss,speed_ms,0,blend_radius_m)
    |   movel([0.295486, -1.278619, -2.636786, -0.796984, 1.570796, 1.866282],accel_mss,speed_ms,0,blend_radius_m)
    |   movel([0.296506, -1.278682, -2.636751, -0.796956, 1.570796, 1.867303],accel_mss,speed_ms,0,blend_radius_m)
    |   movel([0.297837, -1.279317, -2.636390, -0.796683, 1.570796, 1.868633],accel_mss,speed_ms,0,blend_radius_m)
    |   movel([0.298072, -1.279421, -2.636330, -0.796638, 1.570796, 1.868869],accel_mss,speed_ms,0,blend_radius_m)
    |   movel([0.298327, -1.279373, -2.636358, -0.796659, 1.570796, 1.869123],accel_mss,speed_ms,0,blend_radius_m)
    |   movel([0.298659, -1.279143, -2.636488, -0.796757, 1.570796, 1.869456],accel_mss,speed_ms,0,blend_radius_m)
    |   movel([0.300647, -1.277740, -2.637285, -0.797364, 1.570796, 1.871443],accel_mss,speed_ms,0,blend_radius_m)
    |   movel([0.301164, -1.277542, -2.637397, -0.797449, 1.570796, 1.871960],accel_mss,speed_ms,0,blend_radius_m)
    |   movel([0.302128, -1.277538, -2.637400, -0.797451, 1.570796, 1.872924],accel_mss,speed_ms,0,blend_radius_m)
    |   movel([0.302516, -1.277729, -2.637292, -0.797369, 1.570796, 1.873313],accel_mss,speed_ms,0,blend_radius_m)
    |   movel([0.303534, -1.278879, -2.636639, -0.796871, 1.570796, 1.874331],accel_mss,speed_ms,0,blend_radius_m)
    |   movel([0.303710, -1.279014, -2.636562, -0.796813, 1.570796, 1.874507],accel_mss,speed_ms,0,blend_radius_m)
    |   movel([0.304112, -1.278884, -2.636636, -0.796869, 1.570796, 1.874909],accel_mss,speed_ms,0,blend_radius_m)
    |   movel([0.304270, -1.278746, -2.636714, -0.796929, 1.570796, 1.875066],accel_mss,speed_ms,0,blend_radius_m)
    |   movel([0.304601, -1.278282, -2.636978, -0.797129, 1.570796, 1.875398],accel_mss,speed_ms,0,blend_radius_m)
    |   movel([0.304563, -1.277853, -2.637222, -0.797315, 1.570796, 1.875360],accel_mss,speed_ms,0,blend_radius_m)
    |   movel([0.303997, -1.277210, -2.637586, -0.797593, 1.570796, 1.874794],accel_mss,speed_ms,0,blend_radius_m)
    |   movel([0.303742, -1.276998, -2.637706, -0.797685, 1.570796, 1.874539],accel_mss,speed_ms,0,blend_radius_m)
    |   speed_ms = 0.005
    |   movel([0.303742, -1.267659, -2.633242, -0.811488, 1.570796, 1.874539],accel_mss,speed_ms,0,blend_radius_m)
    |   speed_ms = 0.040
    |   movel([0.310187, -1.270451, -2.631677, -0.810261, 1.570796, 1.880984],accel_mss,speed_ms,0,blend_radius_m)
    |   speed_ms = 0.005
    |   movel([0.310187, -1.279776, -2.636128, -0.796485, 1.570796, 1.880984],accel_mss,speed_ms,0,blend_radius_m)
    |   speed_ms = 0.025
    |   movel([0.307945, -1.281298, -2.635259, -0.795831, 1.570796, 1.878742],accel_mss,speed_ms,0,blend_radius_m)
    |   movel([0.307239, -1.281847, -2.634945, -0.795596, 1.570796, 1.878035],accel_mss,speed_ms,0,blend_radius_m)
    |   movel([0.306179, -1.282676, -2.634471, -0.795242, 1.570796, 1.876975],accel_mss,speed_ms,0,blend_radius_m)
    |   movel([0.305530, -1.283080, -2.634239, -0.795070, 1.570796, 1.876327],accel_mss,speed_ms,0,blend_radius_m)
    |   movel([0.305169, -1.283149, -2.634199, -0.795040, 1.570796, 1.875966],accel_mss,speed_ms,0,blend_radius_m)
    |   movel([0.305005, -1.282965, -2.634305, -0.795119, 1.570796, 1.875802],accel_mss,speed_ms,0,blend_radius_m)
    |   movel([0.305156, -1.282578, -2.634527, -0.795284, 1.570796, 1.875952],accel_mss,speed_ms,0,blend_radius_m)
    |   movel([0.305742, -1.281943, -2.634891, -0.795555, 1.570796, 1.876538],accel_mss,speed_ms,0,blend_radius_m)
    |   movel([0.307656, -1.280407, -2.635768, -0.796213, 1.570796, 1.878452],accel_mss,speed_ms,0,blend_radius_m)
    |   movel([0.308166, -1.280045, -2.635975, -0.796369, 1.570796, 1.878962],accel_mss,speed_ms,0,blend_radius_m)
    |   movel([0.309024, -1.279381, -2.636353, -0.796655, 1.570796, 1.879821],accel_mss,speed_ms,0,blend_radius_m)
    |   movel([0.308213, -1.279004, -2.636568, -0.796818, 1.570796, 1.879009],accel_mss,speed_ms,0,blend_radius_m)
    |   movel([0.308069, -1.278762, -2.636705, -0.796922, 1.570796, 1.878866],accel_mss,speed_ms,0,blend_radius_m)
    |   movel([0.308090, -1.278475, -2.636868, -0.797046, 1.570796, 1.878886],accel_mss,speed_ms,0,blend_radius_m)
    |   movel([0.308274, -1.278168, -2.637042, -0.797178, 1.570796, 1.879071],accel_mss,speed_ms,0,blend_radius_m)
    |   movel([0.309211, -1.277368, -2.637496, -0.797525, 1.570796, 1.880008],accel_mss,speed_ms,0,blend_radius_m)
    |   movel([0.310774, -1.276498, -2.637989, -0.797902, 1.570796, 1.881570],accel_mss,speed_ms,0,blend_radius_m)
    |   movel([0.311410, -1.276223, -2.638144, -0.798022, 1.570796, 1.882207],accel_mss,speed_ms,0,blend_radius_m)
    |   movel([0.311806, -1.276156, -2.638182, -0.798051, 1.570796, 1.882602],accel_mss,speed_ms,0,blend_radius_m)
    |   movel([0.311984, -1.276283, -2.638110, -0.797996, 1.570796, 1.882780],accel_mss,speed_ms,0,blend_radius_m)
    |   movel([0.311969, -1.276583, -2.637941, -0.797865, 1.570796, 1.882765],accel_mss,speed_ms,0,blend_radius_m)
    |   movel([0.311630, -1.276996, -2.637707, -0.797686, 1.570796, 1.882426],accel_mss,speed_ms,0,blend_radius_m)
    |   movel([0.311289, -1.277227, -2.637576, -0.797586, 1.570796, 1.882085],accel_mss,speed_ms,0,blend_radius_m)
    |   movel([0.310019, -1.277946, -2.637168, -0.797274, 1.570796, 1.880815],accel_mss,speed_ms,0,blend_radius_m)
    |   movel([0.310117, -1.278213, -2.637017, -0.797159, 1.570796, 1.880913],accel_mss,speed_ms,0,blend_radius_m)
    |   movel([0.310348, -1.278232, -2.637006, -0.797151, 1.570796, 1.881144],accel_mss,speed_ms,0,blend_radius_m)
    |   movel([0.311396, -1.278154, -2.637051, -0.797185, 1.570796, 1.882192],accel_mss,speed_ms,0,blend_radius_m)
    |   movel([0.311633, -1.278208, -2.637020, -0.797161, 1.570796, 1.882430],accel_mss,speed_ms,0,blend_radius_m)
    |   movel([0.311659, -1.278658, -2.636764, -0.796967, 1.570796, 1.882455],accel_mss,speed_ms,0,blend_radius_m)
    |   movel([0.311532, -1.278849, -2.636656, -0.796884, 1.570796, 1.882328],accel_mss,speed_ms,0,blend_radius_m)
    |   movel([0.310779, -1.279421, -2.636330, -0.796638, 1.570796, 1.881575],accel_mss,speed_ms,0,blend_radius_m)
    |   movel([0.310187, -1.279776, -2.636128, -0.796485, 1.570796, 1.880984],accel_mss,speed_ms,0,blend_radius_m)
    |   movel([0.307945, -1.281298, -2.635259, -0.795831, 1.570796, 1.878742],accel_mss,speed_ms,0,blend_radius_m)
    |   movel([0.307496, -1.281648, -2.635060, -0.795682, 1.570796, 1.878292],accel_mss,speed_ms,0,blend_radius_m)
    |   speed_ms = 0.005
    |   movel([0.307496, -1.272333, -2.630617, -0.809439, 1.570796, 1.878292],accel_mss,speed_ms,0,blend_radius_m)
    |   speed_ms = 0.040
    |   movel([0.317906, -1.261503, -2.636658, -0.814228, 1.570796, 1.888702],accel_mss,speed_ms,0,blend_radius_m)
    |   speed_ms = 0.005
    |   movel([0.317906, -1.270874, -2.641149, -0.800365, 1.570796, 1.888702],accel_mss,speed_ms,0,blend_radius_m)
    |   speed_ms = 0.025
    |   movel([0.318381, -1.270685, -2.641255, -0.800449, 1.570796, 1.889177],accel_mss,speed_ms,0,blend_radius_m)
    |   movel([0.318701, -1.270510, -2.641353, -0.800526, 1.570796, 1.889497],accel_mss,speed_ms,0,blend_radius_m)
    |   movel([0.319066, -1.270100, -2.641582, -0.800707, 1.570796, 1.889862],accel_mss,speed_ms,0,blend_radius_m)
    |   movel([0.319113, -1.269763, -2.641769, -0.800856, 1.570796, 1.889909],accel_mss,speed_ms,0,blend_radius_m)
    |   movel([0.318911, -1.269612, -2.641853, -0.800923, 1.570796, 1.889708],accel_mss,speed_ms,0,blend_radius_m)
    |   movel([0.318400, -1.269684, -2.641814, -0.800892, 1.570796, 1.889196],accel_mss,speed_ms,0,blend_radius_m)
    |   movel([0.317542, -1.270002, -2.641637, -0.800751, 1.570796, 1.888338],accel_mss,speed_ms,0,blend_radius_m)
    |   movel([0.316594, -1.270482, -2.641369, -0.800538, 1.570796, 1.887391],accel_mss,speed_ms,0,blend_radius_m)
    |   movel([0.315582, -1.271160, -2.640990, -0.800239, 1.570796, 1.886379],accel_mss,speed_ms,0,blend_radius_m)
    |   movel([0.314756, -1.271843, -2.640608, -0.799938, 1.570796, 1.885552],accel_mss,speed_ms,0,blend_radius_m)
    |   movel([0.314545, -1.272241, -2.640385, -0.799763, 1.570796, 1.885341],accel_mss,speed_ms,0,blend_radius_m)
    |   movel([0.314665, -1.272443, -2.640272, -0.799674, 1.570796, 1.885461],accel_mss,speed_ms,0,blend_radius_m)
    |   movel([0.314965, -1.272458, -2.640263, -0.799668, 1.570796, 1.885762],accel_mss,speed_ms,0,blend_radius_m)
    |   movel([0.315444, -1.272262, -2.640373, -0.799754, 1.570796, 1.886241],accel_mss,speed_ms,0,blend_radius_m)
    |   movel([0.316060, -1.271865, -2.640596, -0.799929, 1.570796, 1.886856],accel_mss,speed_ms,0,blend_radius_m)
    |   movel([0.316470, -1.271594, -2.640747, -0.800048, 1.570796, 1.887267],accel_mss,speed_ms,0,blend_radius_m)
    |   movel([0.317906, -1.270874, -2.641149, -0.800365, 1.570796, 1.888702],accel_mss,speed_ms,0,blend_radius_m)
    |   movel([0.318381, -1.270685, -2.641255, -0.800449, 1.570796, 1.889177],accel_mss,speed_ms,0,blend_radius_m)
    |   movel([0.318701, -1.270510, -2.641353, -0.800526, 1.570796, 1.889497],accel_mss,speed_ms,0,blend_radius_m)
    |   movel([0.319066, -1.270100, -2.641582, -0.800707, 1.570796, 1.889862],accel_mss,speed_ms,0,blend_radius_m)
    |   movel([0.319113, -1.269763, -2.641769, -0.800856, 1.570796, 1.889909],accel_mss,speed_ms,0,blend_radius_m)
    |   movel([0.318911, -1.269612, -2.641853, -0.800923, 1.570796, 1.889708],accel_mss,speed_ms,0,blend_radius_m)
    |   movel([0.318400, -1.269684, -2.641814, -0.800892, 1.570796, 1.889196],accel_mss,speed_ms,0,blend_radius_m)
    |   movel([0.318057, -1.269811, -2.641743, -0.800835, 1.570796, 1.888853],accel_mss,speed_ms,0,blend_radius_m)
    |   speed_ms = 0.005
    |   movel([0.318057, -1.260434, -2.637246, -0.814708, 1.570796, 1.888853],accel_mss,speed_ms,0,blend_radius_m)
    |   speed_ms = 0.040
    |   movel([0.319697, -1.256889, -2.639188, -0.816312, 1.570796, 1.890493],accel_mss,speed_ms,0,blend_radius_m)
    |   speed_ms = 0.005
    |   movel([0.319697, -1.266283, -2.643701, -0.802405, 1.570796, 1.890493],accel_mss,speed_ms,0,blend_radius_m)
    |   speed_ms = 0.025
    |   movel([0.316555, -1.268147, -2.642668, -0.801574, 1.570796, 1.887352],accel_mss,speed_ms,0,blend_radius_m)
    |   movel([0.315703, -1.268699, -2.642362, -0.801329, 1.570796, 1.886499],accel_mss,speed_ms,0,blend_radius_m)
    |   movel([0.315158, -1.268926, -2.642235, -0.801227, 1.570796, 1.885954],accel_mss,speed_ms,0,blend_radius_m)
    |   movel([0.314882, -1.268864, -2.642270, -0.801255, 1.570796, 1.885678],accel_mss,speed_ms,0,blend_radius_m)
    |   movel([0.314820, -1.268562, -2.642438, -0.801389, 1.570796, 1.885617],accel_mss,speed_ms,0,blend_radius_m)
    |   movel([0.315124, -1.268104, -2.642692, -0.801593, 1.570796, 1.885920],accel_mss,speed_ms,0,blend_radius_m)
    |   movel([0.316213, -1.267302, -2.643137, -0.801950, 1.570796, 1.887009],accel_mss,speed_ms,0,blend_radius_m)
    |   movel([0.317715, -1.266349, -2.643665, -0.802376, 1.570796, 1.888511],accel_mss,speed_ms,0,blend_radius_m)
    |   movel([0.320749, -1.264720, -2.644564, -0.803105, 1.570796, 1.891546],accel_mss,speed_ms,0,blend_radius_m)
    |   movel([0.321427, -1.264494, -2.644688, -0.803207, 1.570796, 1.892223],accel_mss,speed_ms,0,blend_radius_m)
    |   movel([0.321734, -1.264574, -2.644644, -0.803171, 1.570796, 1.892530],accel_mss,speed_ms,0,blend_radius_m)
    |   movel([0.321765, -1.264894, -2.644468, -0.803027, 1.570796, 1.892561],accel_mss,speed_ms,0,blend_radius_m)
    |   movel([0.321607, -1.265117, -2.644345, -0.802927, 1.570796, 1.892403],accel_mss,speed_ms,0,blend_radius_m)
    |   movel([0.321229, -1.265405, -2.644186, -0.802798, 1.570796, 1.892026],accel_mss,speed_ms,0,blend_radius_m)
    |   movel([0.319697, -1.266283, -2.643701, -0.802405, 1.570796, 1.890493],accel_mss,speed_ms,0,blend_radius_m)
    |   movel([0.316872, -1.267961, -2.642771, -0.801656, 1.570796, 1.887668],accel_mss,speed_ms,0,blend_radius_m)
    |   speed_ms = 0.005
    |   movel([0.316872, -1.258575, -2.638267, -0.815547, 1.570796, 1.887668],accel_mss,speed_ms,0,blend_radius_m)
    |   speed_ms = 0.040
    |   movel([0.320388, -1.258483, -2.638317, -0.815589, 1.570796, 1.891184],accel_mss,speed_ms,0,blend_radius_m)
    |   speed_ms = 0.005
    |   movel([0.320388, -1.267869, -2.642822, -0.801697, 1.570796, 1.891184],accel_mss,speed_ms,0,blend_radius_m)
    |   speed_ms = 0.025
    |   movel([0.320776, -1.267555, -2.642997, -0.801837, 1.570796, 1.891573],accel_mss,speed_ms,0,blend_radius_m)
    |   movel([0.320923, -1.267216, -2.643185, -0.801988, 1.570796, 1.891720],accel_mss,speed_ms,0,blend_radius_m)
    |   movel([0.320765, -1.266975, -2.643318, -0.802096, 1.570796, 1.891561],accel_mss,speed_ms,0,blend_radius_m)
    |   movel([0.320356, -1.266938, -2.643339, -0.802112, 1.570796, 1.891152],accel_mss,speed_ms,0,blend_radius_m)
    |   movel([0.319050, -1.267311, -2.643132, -0.801946, 1.570796, 1.889847],accel_mss,speed_ms,0,blend_radius_m)
    |   movel([0.317372, -1.268122, -2.642682, -0.801585, 1.570796, 1.888168],accel_mss,speed_ms,0,blend_radius_m)
    |   movel([0.315857, -1.269052, -2.642165, -0.801172, 1.570796, 1.886653],accel_mss,speed_ms,0,blend_radius_m)
    |   movel([0.315533, -1.269350, -2.642000, -0.801040, 1.570796, 1.886329],accel_mss,speed_ms,0,blend_radius_m)
    |   movel([0.315336, -1.269703, -2.641803, -0.800883, 1.570796, 1.886132],accel_mss,speed_ms,0,blend_radius_m)
    |   movel([0.315327, -1.270028, -2.641622, -0.800739, 1.570796, 1.886124],accel_mss,speed_ms,0,blend_radius_m)
    |   movel([0.315536, -1.270129, -2.641566, -0.800695, 1.570796, 1.886332],accel_mss,speed_ms,0,blend_radius_m)
    |   movel([0.316012, -1.269966, -2.641657, -0.800767, 1.570796, 1.886809],accel_mss,speed_ms,0,blend_radius_m)
    |   movel([0.317328, -1.269196, -2.642085, -0.801108, 1.570796, 1.888125],accel_mss,speed_ms,0,blend_radius_m)
    |   movel([0.317934, -1.268881, -2.642261, -0.801248, 1.570796, 1.888730],accel_mss,speed_ms,0,blend_radius_m)
    |   movel([0.320388, -1.267869, -2.642822, -0.801697, 1.570796, 1.891184],accel_mss,speed_ms,0,blend_radius_m)
    |   movel([0.320776, -1.267555, -2.642997, -0.801837, 1.570796, 1.891573],accel_mss,speed_ms,0,blend_radius_m)
    |   movel([0.320923, -1.267216, -2.643185, -0.801988, 1.570796, 1.891720],accel_mss,speed_ms,0,blend_radius_m)
    |   movel([0.320765, -1.266975, -2.643318, -0.802096, 1.570796, 1.891561],accel_mss,speed_ms,0,blend_radius_m)
    |   movel([0.320356, -1.266938, -2.643339, -0.802112, 1.570796, 1.891152],accel_mss,speed_ms,0,blend_radius_m)
    |   movel([0.319149, -1.267281, -2.643148, -0.801959, 1.570796, 1.889945],accel_mss,speed_ms,0,blend_radius_m)
    |   speed_ms = 0.005
    |   movel([0.319149, -1.257892, -2.638640, -0.815857, 1.570796, 1.889945],accel_mss,speed_ms,0,blend_radius_m)
    |   speed_ms = 0.040
    |   movel([0.342305, -1.256445, -2.639430, -0.816513, 1.570796, 1.913101],accel_mss,speed_ms,0,blend_radius_m)
    |   speed_ms = 0.005
    |   movel([0.342305, -1.265842, -2.643945, -0.802602, 1.570796, 1.913101],accel_mss,speed_ms,0,blend_radius_m)
    |   speed_ms = 0.025
    |   movel([0.342098, -1.265915, -2.643904, -0.802570, 1.570796, 1.912894],accel_mss,speed_ms,0,blend_radius_m)
    |   movel([0.340491, -1.266862, -2.643381, -0.802146, 1.570796, 1.911288],accel_mss,speed_ms,0,blend_radius_m)
    |   movel([0.336963, -1.269040, -2.642172, -0.801177, 1.570796, 1.907759],accel_mss,speed_ms,0,blend_radius_m)
    |   movel([0.336711, -1.269272, -2.642043, -0.801074, 1.570796, 1.907507],accel_mss,speed_ms,0,blend_radius_m)
    |   movel([0.336460, -1.269923, -2.641680, -0.800786, 1.570796, 1.907256],accel_mss,speed_ms,0,blend_radius_m)
    |   movel([0.336394, -1.270253, -2.641497, -0.800640, 1.570796, 1.907190],accel_mss,speed_ms,0,blend_radius_m)
    |   movel([0.335810, -1.272745, -2.640102, -0.799541, 1.570796, 1.906606],accel_mss,speed_ms,0,blend_radius_m)
    |   movel([0.334250, -1.273578, -2.639635, -0.799176, 1.570796, 1.905046],accel_mss,speed_ms,0,blend_radius_m)
    |   movel([0.331241, -1.275069, -2.638796, -0.798524, 1.570796, 1.902037],accel_mss,speed_ms,0,blend_radius_m)
    |   movel([0.330813, -1.275442, -2.638585, -0.798362, 1.570796, 1.901609],accel_mss,speed_ms,0,blend_radius_m)
    |   movel([0.330450, -1.276018, -2.638260, -0.798111, 1.570796, 1.901246],accel_mss,speed_ms,0,blend_radius_m)
    |   movel([0.329947, -1.277140, -2.637625, -0.797623, 1.570796, 1.900744],accel_mss,speed_ms,0,blend_radius_m)
    |   movel([0.329287, -1.278475, -2.636868, -0.797046, 1.570796, 1.900084],accel_mss,speed_ms,0,blend_radius_m)
    |   movel([0.328562, -1.279472, -2.636301, -0.796616, 1.570796, 1.899359],accel_mss,speed_ms,0,blend_radius_m)
    |   movel([0.327678, -1.280249, -2.635858, -0.796281, 1.570796, 1.898474],accel_mss,speed_ms,0,blend_radius_m)
    |   movel([0.326542, -1.280909, -2.635482, -0.795998, 1.570796, 1.897338],accel_mss,speed_ms,0,blend_radius_m)
    |   movel([0.326144, -1.281152, -2.635343, -0.795894, 1.570796, 1.896940],accel_mss,speed_ms,0,blend_radius_m)
    |   movel([0.325887, -1.281432, -2.635183, -0.795774, 1.570796, 1.896683],accel_mss,speed_ms,0,blend_radius_m)
    |   movel([0.325103, -1.283251, -2.634141, -0.794997, 1.570796, 1.895899],accel_mss,speed_ms,0,blend_radius_m)
    |   movel([0.324590, -1.284623, -2.633352, -0.794414, 1.570796, 1.895386],accel_mss,speed_ms,0,blend_radius_m)
    |   movel([0.324435, -1.285304, -2.632960, -0.794125, 1.570796, 1.895231],accel_mss,speed_ms,0,blend_radius_m)
    |   movel([0.324599, -1.285346, -2.632936, -0.794107, 1.570796, 1.895395],accel_mss,speed_ms,0,blend_radius_m)
    |   movel([0.324950, -1.285005, -2.633132, -0.794252, 1.570796, 1.895746],accel_mss,speed_ms,0,blend_radius_m)
    |   movel([0.326095, -1.283460, -2.634021, -0.794908, 1.570796, 1.896892],accel_mss,speed_ms,0,blend_radius_m)
    |   movel([0.328453, -1.280507, -2.635711, -0.796171, 1.570796, 1.899249],accel_mss,speed_ms,0,blend_radius_m)
    |   movel([0.329314, -1.279540, -2.636262, -0.796586, 1.570796, 1.900110],accel_mss,speed_ms,0,blend_radius_m)
    |   movel([0.331878, -1.277185, -2.637600, -0.797604, 1.570796, 1.902674],accel_mss,speed_ms,0,blend_radius_m)
    |   movel([0.333689, -1.275680, -2.638451, -0.798258, 1.570796, 1.904485],accel_mss,speed_ms,0,blend_radius_m)
    |   movel([0.336596, -1.273329, -2.639775, -0.799285, 1.570796, 1.907392],accel_mss,speed_ms,0,blend_radius_m)
    |   movel([0.337272, -1.272571, -2.640200, -0.799618, 1.570796, 1.908068],accel_mss,speed_ms,0,blend_radius_m)
    |   movel([0.337811, -1.271674, -2.640702, -0.800012, 1.570796, 1.908607],accel_mss,speed_ms,0,blend_radius_m)
    |   movel([0.338397, -1.270330, -2.641453, -0.800605, 1.570796, 1.909193],accel_mss,speed_ms,0,blend_radius_m)
    |   movel([0.339374, -1.268074, -2.642709, -0.801606, 1.570796, 1.910170],accel_mss,speed_ms,0,blend_radius_m)
    |   movel([0.339665, -1.267770, -2.642878, -0.801742, 1.570796, 1.910462],accel_mss,speed_ms,0,blend_radius_m)
    |   movel([0.340001, -1.267655, -2.642941, -0.801793, 1.570796, 1.910798],accel_mss,speed_ms,0,blend_radius_m)
    |   movel([0.340202, -1.267710, -2.642911, -0.801768, 1.570796, 1.910999],accel_mss,speed_ms,0,blend_radius_m)
    |   movel([0.340260, -1.268163, -2.642659, -0.801566, 1.570796, 1.911056],accel_mss,speed_ms,0,blend_radius_m)
    |   movel([0.340097, -1.268815, -2.642297, -0.801277, 1.570796, 1.910894],accel_mss,speed_ms,0,blend_radius_m)
    |   movel([0.339787, -1.269967, -2.641656, -0.800766, 1.570796, 1.910583],accel_mss,speed_ms,0,blend_radius_m)
    |   movel([0.340392, -1.269168, -2.642101, -0.801120, 1.570796, 1.911189],accel_mss,speed_ms,0,blend_radius_m)
    |   movel([0.342216, -1.266344, -2.643667, -0.802378, 1.570796, 1.913012],accel_mss,speed_ms,0,blend_radius_m)
    |   movel([0.342407, -1.265942, -2.643890, -0.802558, 1.570796, 1.913204],accel_mss,speed_ms,0,blend_radius_m)
    |   movel([0.342305, -1.265842, -2.643945, -0.802602, 1.570796, 1.913101],accel_mss,speed_ms,0,blend_radius_m)
    |   movel([0.342098, -1.265915, -2.643904, -0.802570, 1.570796, 1.912894],accel_mss,speed_ms,0,blend_radius_m)
    |   movel([0.340491, -1.266862, -2.643381, -0.802146, 1.570796, 1.911288],accel_mss,speed_ms,0,blend_radius_m)
    |   movel([0.339477, -1.267486, -2.643035, -0.801868, 1.570796, 1.910274],accel_mss,speed_ms,0,blend_radius_m)
    |   speed_ms = 0.005
    |   movel([0.339477, -1.258098, -2.638528, -0.815763, 1.570796, 1.910274],accel_mss,speed_ms,0,blend_radius_m)
    |   speed_ms = 0.040
    |   movel([0.320993, -1.272658, -2.630434, -0.809298, 1.570796, 1.891789],accel_mss,speed_ms,0,blend_radius_m)
    |   speed_ms = 0.005
    |   movel([0.320993, -1.281971, -2.634875, -0.795543, 1.570796, 1.891789],accel_mss,speed_ms,0,blend_radius_m)
    |   speed_ms = 0.025
    |   movel([0.316988, -1.287635, -2.631612, -0.793142, 1.570796, 1.887784],accel_mss,speed_ms,0,blend_radius_m)
    |   movel([0.316395, -1.288468, -2.631129, -0.792792, 1.570796, 1.887191],accel_mss,speed_ms,0,blend_radius_m)
    |   movel([0.315808, -1.289374, -2.630603, -0.792413, 1.570796, 1.886604],accel_mss,speed_ms,0,blend_radius_m)
    |   movel([0.315747, -1.289880, -2.630308, -0.792201, 1.570796, 1.886543],accel_mss,speed_ms,0,blend_radius_m)
    |   movel([0.316142, -1.291767, -2.629206, -0.791415, 1.570796, 1.886939],accel_mss,speed_ms,0,blend_radius_m)
    |   movel([0.316420, -1.292372, -2.628852, -0.791164, 1.570796, 1.887216],accel_mss,speed_ms,0,blend_radius_m)
    |   movel([0.317118, -1.293053, -2.628454, -0.790883, 1.570796, 1.887915],accel_mss,speed_ms,0,blend_radius_m)
    |   movel([0.317362, -1.293182, -2.628378, -0.790829, 1.570796, 1.888158],accel_mss,speed_ms,0,blend_radius_m)
    |   movel([0.317767, -1.293446, -2.628223, -0.790720, 1.570796, 1.888564],accel_mss,speed_ms,0,blend_radius_m)
    |   movel([0.317796, -1.293609, -2.628127, -0.790653, 1.570796, 1.888593],accel_mss,speed_ms,0,blend_radius_m)
    |   movel([0.317736, -1.293818, -2.628004, -0.790567, 1.570796, 1.888533],accel_mss,speed_ms,0,blend_radius_m)
    |   movel([0.317454, -1.294161, -2.627803, -0.790425, 1.570796, 1.888251],accel_mss,speed_ms,0,blend_radius_m)
    |   movel([0.317075, -1.294326, -2.627706, -0.790357, 1.570796, 1.887871],accel_mss,speed_ms,0,blend_radius_m)
    |   movel([0.316601, -1.294268, -2.627740, -0.790381, 1.570796, 1.887397],accel_mss,speed_ms,0,blend_radius_m)
    |   movel([0.316051, -1.293981, -2.627908, -0.790499, 1.570796, 1.886847],accel_mss,speed_ms,0,blend_radius_m)
    |   movel([0.315348, -1.293224, -2.628353, -0.790812, 1.570796, 1.886144],accel_mss,speed_ms,0,blend_radius_m)
    |   movel([0.314820, -1.291942, -2.629104, -0.791343, 1.570796, 1.885616],accel_mss,speed_ms,0,blend_radius_m)
    |   movel([0.314555, -1.290535, -2.629926, -0.791928, 1.570796, 1.885351],accel_mss,speed_ms,0,blend_radius_m)
    |   movel([0.314708, -1.289398, -2.630589, -0.792403, 1.570796, 1.885505],accel_mss,speed_ms,0,blend_radius_m)
    |   movel([0.314869, -1.289065, -2.630782, -0.792542, 1.570796, 1.885666],accel_mss,speed_ms,0,blend_radius_m)
    |   movel([0.316629, -1.286570, -2.632229, -0.793590, 1.570796, 1.887425],accel_mss,speed_ms,0,blend_radius_m)
    |   movel([0.318018, -1.284686, -2.633316, -0.794387, 1.570796, 1.888814],accel_mss,speed_ms,0,blend_radius_m)
    |   movel([0.321170, -1.280134, -2.635924, -0.796331, 1.570796, 1.891966],accel_mss,speed_ms,0,blend_radius_m)
    |   movel([0.321478, -1.279523, -2.636272, -0.796594, 1.570796, 1.892275],accel_mss,speed_ms,0,blend_radius_m)
    |   movel([0.321643, -1.279254, -2.636426, -0.796710, 1.570796, 1.892440],accel_mss,speed_ms,0,blend_radius_m)
    |   movel([0.321947, -1.278993, -2.636574, -0.796822, 1.570796, 1.892743],accel_mss,speed_ms,0,blend_radius_m)
    |   movel([0.322286, -1.278817, -2.636674, -0.796898, 1.570796, 1.893083],accel_mss,speed_ms,0,blend_radius_m)
    |   movel([0.322545, -1.278797, -2.636685, -0.796907, 1.570796, 1.893341],accel_mss,speed_ms,0,blend_radius_m)
    |   movel([0.322683, -1.279013, -2.636563, -0.796814, 1.570796, 1.893479],accel_mss,speed_ms,0,blend_radius_m)
    |   movel([0.322549, -1.279463, -2.636306, -0.796620, 1.570796, 1.893345],accel_mss,speed_ms,0,blend_radius_m)
    |   movel([0.320993, -1.281971, -2.634875, -0.795543, 1.570796, 1.891789],accel_mss,speed_ms,0,blend_radius_m)
    |   movel([0.319159, -1.284560, -2.633389, -0.794441, 1.570796, 1.889955],accel_mss,speed_ms,0,blend_radius_m)
    |   speed_ms = 0.005
    |   movel([0.319159, -1.275261, -2.628959, -0.808169, 1.570796, 1.889955],accel_mss,speed_ms,0,blend_radius_m)
    |   speed_ms = 0.040
    |   movel([0.311817, -1.274901, -2.629163, -0.808325, 1.570796, 1.882613],accel_mss,speed_ms,0,blend_radius_m)
    |   speed_ms = 0.005
    |   movel([0.311817, -1.284202, -2.633594, -0.794592, 1.570796, 1.882613],accel_mss,speed_ms,0,blend_radius_m)
    |   speed_ms = 0.025
    |   movel([0.312123, -1.284010, -2.633705, -0.794674, 1.570796, 1.882920],accel_mss,speed_ms,0,blend_radius_m)
    |   movel([0.312434, -1.283540, -2.633975, -0.794874, 1.570796, 1.883230],accel_mss,speed_ms,0,blend_radius_m)
    |   movel([0.312386, -1.283350, -2.634084, -0.794955, 1.570796, 1.883182],accel_mss,speed_ms,0,blend_radius_m)
    |   movel([0.312161, -1.283224, -2.634157, -0.795009, 1.570796, 1.882957],accel_mss,speed_ms,0,blend_radius_m)
    |   movel([0.311843, -1.283250, -2.634142, -0.794998, 1.570796, 1.882639],accel_mss,speed_ms,0,blend_radius_m)
    |   movel([0.309502, -1.283994, -2.633714, -0.794681, 1.570796, 1.880298],accel_mss,speed_ms,0,blend_radius_m)
    |   movel([0.306967, -1.284934, -2.633173, -0.794282, 1.570796, 1.877763],accel_mss,speed_ms,0,blend_radius_m)
    |   movel([0.304712, -1.285945, -2.632590, -0.793854, 1.570796, 1.875508],accel_mss,speed_ms,0,blend_radius_m)
    |   movel([0.304096, -1.286245, -2.632417, -0.793727, 1.570796, 1.874893],accel_mss,speed_ms,0,blend_radius_m)
    |   movel([0.303072, -1.286689, -2.632160, -0.793540, 1.570796, 1.873868],accel_mss,speed_ms,0,blend_radius_m)
    |   movel([0.311710, -1.280608, -2.635654, -0.796127, 1.570796, 1.882506],accel_mss,speed_ms,0,blend_radius_m)
    |   movel([0.312421, -1.279966, -2.636020, -0.796403, 1.570796, 1.883218],accel_mss,speed_ms,0,blend_radius_m)
    |   movel([0.312621, -1.279559, -2.636252, -0.796578, 1.570796, 1.883418],accel_mss,speed_ms,0,blend_radius_m)
    |   movel([0.312461, -1.279312, -2.636393, -0.796685, 1.570796, 1.883257],accel_mss,speed_ms,0,blend_radius_m)
    |   movel([0.312167, -1.279321, -2.636387, -0.796681, 1.570796, 1.882963],accel_mss,speed_ms,0,blend_radius_m)
    |   movel([0.311845, -1.279472, -2.636301, -0.796616, 1.570796, 1.882641],accel_mss,speed_ms,0,blend_radius_m)
    |   movel([0.306835, -1.282923, -2.634329, -0.795137, 1.570796, 1.877631],accel_mss,speed_ms,0,blend_radius_m)
    |   movel([0.301566, -1.286656, -2.632179, -0.793554, 1.570796, 1.872363],accel_mss,speed_ms,0,blend_radius_m)
    |   movel([0.296386, -1.290477, -2.629960, -0.791952, 1.570796, 1.867183],accel_mss,speed_ms,0,blend_radius_m)
    |   movel([0.294549, -1.291895, -2.629132, -0.791362, 1.570796, 1.865346],accel_mss,speed_ms,0,blend_radius_m)
    |   movel([0.293631, -1.292725, -2.628646, -0.791018, 1.570796, 1.864428],accel_mss,speed_ms,0,blend_radius_m)
    |   movel([0.293344, -1.293200, -2.628367, -0.790822, 1.570796, 1.864140],accel_mss,speed_ms,0,blend_radius_m)
    |   movel([0.293473, -1.293471, -2.628208, -0.790710, 1.570796, 1.864269],accel_mss,speed_ms,0,blend_radius_m)
    |   movel([0.293657, -1.293435, -2.628229, -0.790725, 1.570796, 1.864453],accel_mss,speed_ms,0,blend_radius_m)
    |   movel([0.296401, -1.291747, -2.629218, -0.791424, 1.570796, 1.867197],accel_mss,speed_ms,0,blend_radius_m)
    |   movel([0.300069, -1.289456, -2.630555, -0.792378, 1.570796, 1.870865],accel_mss,speed_ms,0,blend_radius_m)
    |   movel([0.303670, -1.287486, -2.631699, -0.793204, 1.570796, 1.874467],accel_mss,speed_ms,0,blend_radius_m)
    |   movel([0.307041, -1.285916, -2.632607, -0.793866, 1.570796, 1.877837],accel_mss,speed_ms,0,blend_radius_m)
    |   movel([0.311817, -1.284202, -2.633594, -0.794592, 1.570796, 1.882613],accel_mss,speed_ms,0,blend_radius_m)
    |   movel([0.312123, -1.284010, -2.633705, -0.794674, 1.570796, 1.882920],accel_mss,speed_ms,0,blend_radius_m)
    |   movel([0.312434, -1.283540, -2.633975, -0.794874, 1.570796, 1.883230],accel_mss,speed_ms,0,blend_radius_m)
    |   movel([0.312386, -1.283350, -2.634084, -0.794955, 1.570796, 1.883182],accel_mss,speed_ms,0,blend_radius_m)
    |   movel([0.312161, -1.283224, -2.634157, -0.795009, 1.570796, 1.882957],accel_mss,speed_ms,0,blend_radius_m)
    |   movel([0.311843, -1.283250, -2.634142, -0.794998, 1.570796, 1.882639],accel_mss,speed_ms,0,blend_radius_m)
    |   movel([0.310788, -1.283583, -2.633950, -0.794856, 1.570796, 1.881584],accel_mss,speed_ms,0,blend_radius_m)
    |   speed_ms = 0.005
    |   movel([0.310788, -1.274279, -2.629516, -0.808594, 1.570796, 1.881584],accel_mss,speed_ms,0,blend_radius_m)
    |   speed_ms = 0.040
    |   movel([0.323269, -1.277933, -2.627437, -0.807020, 1.570796, 1.894066],accel_mss,speed_ms,0,blend_radius_m)
    |   speed_ms = 0.005
    |   movel([0.323269, -1.287217, -2.631854, -0.793317, 1.570796, 1.894066],accel_mss,speed_ms,0,blend_radius_m)
    |   speed_ms = 0.025
    |   movel([0.322794, -1.287491, -2.631696, -0.793202, 1.570796, 1.893591],accel_mss,speed_ms,0,blend_radius_m)
    |   movel([0.322568, -1.287543, -2.631665, -0.793180, 1.570796, 1.893364],accel_mss,speed_ms,0,blend_radius_m)
    |   movel([0.322017, -1.287538, -2.631668, -0.793182, 1.570796, 1.892813],accel_mss,speed_ms,0,blend_radius_m)
    |   movel([0.321877, -1.287650, -2.631604, -0.793136, 1.570796, 1.892674],accel_mss,speed_ms,0,blend_radius_m)
    |   movel([0.321851, -1.288812, -2.630929, -0.792648, 1.570796, 1.892647],accel_mss,speed_ms,0,blend_radius_m)
    |   movel([0.321878, -1.289430, -2.630570, -0.792389, 1.570796, 1.892674],accel_mss,speed_ms,0,blend_radius_m)
    |   movel([0.321928, -1.289619, -2.630460, -0.792310, 1.570796, 1.892725],accel_mss,speed_ms,0,blend_radius_m)
    |   movel([0.323540, -1.287177, -2.631878, -0.793334, 1.570796, 1.894337],accel_mss,speed_ms,0,blend_radius_m)
    |   movel([0.323606, -1.287022, -2.631967, -0.793399, 1.570796, 1.894402],accel_mss,speed_ms,0,blend_radius_m)
    |   movel([0.323269, -1.287217, -2.631854, -0.793317, 1.570796, 1.894066],accel_mss,speed_ms,0,blend_radius_m)
    |   movel([0.322794, -1.287491, -2.631696, -0.793202, 1.570796, 1.893591],accel_mss,speed_ms,0,blend_radius_m)
    |   movel([0.322568, -1.287543, -2.631665, -0.793180, 1.570796, 1.893364],accel_mss,speed_ms,0,blend_radius_m)
    |   movel([0.322017, -1.287538, -2.631668, -0.793182, 1.570796, 1.892813],accel_mss,speed_ms,0,blend_radius_m)
    |   movel([0.321877, -1.287650, -2.631604, -0.793136, 1.570796, 1.892674],accel_mss,speed_ms,0,blend_radius_m)
    |   movel([0.321850, -1.288785, -2.630945, -0.792659, 1.570796, 1.892646],accel_mss,speed_ms,0,blend_radius_m)
    |   speed_ms = 0.005
    |   movel([0.321850, -1.279509, -2.626535, -0.806346, 1.570796, 1.892646],accel_mss,speed_ms,0,blend_radius_m)
    |   speed_ms = 0.040
    |   movel([0.314734, -1.287909, -2.621674, -0.802806, 1.570796, 1.885530],accel_mss,speed_ms,0,blend_radius_m)
    |   speed_ms = 0.005
    |   movel([0.314734, -1.297139, -2.626046, -0.789204, 1.570796, 1.885530],accel_mss,speed_ms,0,blend_radius_m)
    |   speed_ms = 0.025
    |   movel([0.315184, -1.296849, -2.626218, -0.789322, 1.570796, 1.885980],accel_mss,speed_ms,0,blend_radius_m)
    |   movel([0.315360, -1.296419, -2.626472, -0.789498, 1.570796, 1.886156],accel_mss,speed_ms,0,blend_radius_m)
    |   movel([0.315168, -1.295772, -2.626854, -0.789763, 1.570796, 1.885965],accel_mss,speed_ms,0,blend_radius_m)
    |   movel([0.314017, -1.294219, -2.627768, -0.790401, 1.570796, 1.884813],accel_mss,speed_ms,0,blend_radius_m)
    |   movel([0.313315, -1.293623, -2.628119, -0.790647, 1.570796, 1.884111],accel_mss,speed_ms,0,blend_radius_m)
    |   movel([0.311218, -1.292395, -2.628839, -0.791155, 1.570796, 1.882015],accel_mss,speed_ms,0,blend_radius_m)
    |   movel([0.310953, -1.292206, -2.628950, -0.791233, 1.570796, 1.881749],accel_mss,speed_ms,0,blend_radius_m)
    |   movel([0.310711, -1.291884, -2.629138, -0.791367, 1.570796, 1.881507],accel_mss,speed_ms,0,blend_radius_m)
    |   movel([0.310760, -1.291671, -2.629263, -0.791455, 1.570796, 1.881557],accel_mss,speed_ms,0,blend_radius_m)
    |   movel([0.311957, -1.289196, -2.630706, -0.792487, 1.570796, 1.882753],accel_mss,speed_ms,0,blend_radius_m)
    |   movel([0.313206, -1.286796, -2.632098, -0.793495, 1.570796, 1.884002],accel_mss,speed_ms,0,blend_radius_m)
    |   movel([0.314487, -1.285737, -2.632710, -0.793942, 1.570796, 1.885284],accel_mss,speed_ms,0,blend_radius_m)
    |   movel([0.315483, -1.284828, -2.633234, -0.794327, 1.570796, 1.886280],accel_mss,speed_ms,0,blend_radius_m)
    |   movel([0.316379, -1.283834, -2.633806, -0.794749, 1.570796, 1.887175],accel_mss,speed_ms,0,blend_radius_m)
    |   movel([0.317174, -1.282752, -2.634427, -0.795210, 1.570796, 1.887970],accel_mss,speed_ms,0,blend_radius_m)
    |   movel([0.318245, -1.280807, -2.635540, -0.796042, 1.570796, 1.889041],accel_mss,speed_ms,0,blend_radius_m)
    |   movel([0.318369, -1.280358, -2.635796, -0.796234, 1.570796, 1.889165],accel_mss,speed_ms,0,blend_radius_m)
    |   movel([0.318281, -1.280137, -2.635922, -0.796329, 1.570796, 1.889077],accel_mss,speed_ms,0,blend_radius_m)
    |   movel([0.317998, -1.280086, -2.635952, -0.796352, 1.570796, 1.888794],accel_mss,speed_ms,0,blend_radius_m)
    |   movel([0.317788, -1.280161, -2.635909, -0.796319, 1.570796, 1.888584],accel_mss,speed_ms,0,blend_radius_m)
    |   movel([0.317594, -1.280310, -2.635824, -0.796255, 1.570796, 1.888391],accel_mss,speed_ms,0,blend_radius_m)
    |   movel([0.316528, -1.282011, -2.634852, -0.795526, 1.570796, 1.887325],accel_mss,speed_ms,0,blend_radius_m)
    |   movel([0.316076, -1.282711, -2.634451, -0.795227, 1.570796, 1.886872],accel_mss,speed_ms,0,blend_radius_m)
    |   movel([0.315050, -1.283982, -2.633721, -0.794686, 1.570796, 1.885846],accel_mss,speed_ms,0,blend_radius_m)
    |   movel([0.314680, -1.284374, -2.633495, -0.794519, 1.570796, 1.885476],accel_mss,speed_ms,0,blend_radius_m)
    |   movel([0.313597, -1.285322, -2.632949, -0.794118, 1.570796, 1.884394],accel_mss,speed_ms,0,blend_radius_m)
    |   movel([0.312972, -1.285832, -2.632655, -0.793902, 1.570796, 1.883768],accel_mss,speed_ms,0,blend_radius_m)
    |   movel([0.312430, -1.286494, -2.632273, -0.793622, 1.570796, 1.883226],accel_mss,speed_ms,0,blend_radius_m)
    |   movel([0.311798, -1.287538, -2.631668, -0.793182, 1.570796, 1.882594],accel_mss,speed_ms,0,blend_radius_m)
    |   movel([0.309350, -1.292270, -2.628912, -0.791207, 1.570796, 1.880146],accel_mss,speed_ms,0,blend_radius_m)
    |   movel([0.309566, -1.292711, -2.628654, -0.791024, 1.570796, 1.880363],accel_mss,speed_ms,0,blend_radius_m)
    |   movel([0.310550, -1.293526, -2.628176, -0.790687, 1.570796, 1.881346],accel_mss,speed_ms,0,blend_radius_m)
    |   movel([0.311050, -1.293811, -2.628008, -0.790569, 1.570796, 1.881846],accel_mss,speed_ms,0,blend_radius_m)
    |   movel([0.312964, -1.295097, -2.627252, -0.790040, 1.570796, 1.883760],accel_mss,speed_ms,0,blend_radius_m)
    |   movel([0.313595, -1.295788, -2.626844, -0.789756, 1.570796, 1.884392],accel_mss,speed_ms,0,blend_radius_m)
    |   movel([0.314171, -1.296856, -2.626214, -0.789319, 1.570796, 1.884968],accel_mss,speed_ms,0,blend_radius_m)
    |   movel([0.314336, -1.297059, -2.626094, -0.789237, 1.570796, 1.885133],accel_mss,speed_ms,0,blend_radius_m)
    |   movel([0.314734, -1.297139, -2.626046, -0.789204, 1.570796, 1.885530],accel_mss,speed_ms,0,blend_radius_m)
    |   movel([0.315184, -1.296849, -2.626218, -0.789322, 1.570796, 1.885980],accel_mss,speed_ms,0,blend_radius_m)
    |   movel([0.315360, -1.296419, -2.626472, -0.789498, 1.570796, 1.886156],accel_mss,speed_ms,0,blend_radius_m)
    |   movel([0.315168, -1.295772, -2.626854, -0.789763, 1.570796, 1.885965],accel_mss,speed_ms,0,blend_radius_m)
    |   movel([0.314744, -1.295199, -2.627192, -0.789998, 1.570796, 1.885541],accel_mss,speed_ms,0,blend_radius_m)
    |   speed_ms = 0.005
    |   movel([0.314744, -1.285959, -2.622810, -0.803620, 1.570796, 1.885541],accel_mss,speed_ms,0,blend_radius_m)
    |   speed_ms = 0.040
    |   movel([0.304596, -1.282856, -2.624608, -0.804924, 1.570796, 1.875393],accel_mss,speed_ms,0,blend_radius_m)
    |   speed_ms = 0.005
    |   movel([0.304596, -1.292114, -2.629003, -0.791271, 1.570796, 1.875393],accel_mss,speed_ms,0,blend_radius_m)
    |   speed_ms = 0.025
    |   movel([0.301176, -1.294538, -2.627581, -0.790270, 1.570796, 1.871973],accel_mss,speed_ms,0,blend_radius_m)
    |   movel([0.297779, -1.297082, -2.626080, -0.789227, 1.570796, 1.868575],accel_mss,speed_ms,0,blend_radius_m)
    |   movel([0.291017, -1.302549, -2.622826, -0.787014, 1.570796, 1.861813],accel_mss,speed_ms,0,blend_radius_m)
    |   movel([0.289582, -1.303752, -2.622105, -0.786532, 1.570796, 1.860378],accel_mss,speed_ms,0,blend_radius_m)
    |   movel([0.287255, -1.305624, -2.620979, -0.785786, 1.570796, 1.858052],accel_mss,speed_ms,0,blend_radius_m)
    |   movel([0.287048, -1.305719, -2.620921, -0.785749, 1.570796, 1.857844],accel_mss,speed_ms,0,blend_radius_m)
    |   movel([0.286760, -1.305582, -2.621004, -0.785803, 1.570796, 1.857557],accel_mss,speed_ms,0,blend_radius_m)
    |   movel([0.286728, -1.305476, -2.621068, -0.785845, 1.570796, 1.857524],accel_mss,speed_ms,0,blend_radius_m)
    |   movel([0.286851, -1.304841, -2.621450, -0.786098, 1.570796, 1.857648],accel_mss,speed_ms,0,blend_radius_m)
    |   movel([0.287297, -1.304200, -2.621836, -0.786353, 1.570796, 1.858093],accel_mss,speed_ms,0,blend_radius_m)
    |   movel([0.302557, -1.288940, -2.630855, -0.792594, 1.570796, 1.873353],accel_mss,speed_ms,0,blend_radius_m)
    |   movel([0.303302, -1.288390, -2.631175, -0.792825, 1.570796, 1.874098],accel_mss,speed_ms,0,blend_radius_m)
    |   movel([0.304097, -1.288114, -2.631334, -0.792940, 1.570796, 1.874893],accel_mss,speed_ms,0,blend_radius_m)
    |   movel([0.304363, -1.288257, -2.631252, -0.792881, 1.570796, 1.875159],accel_mss,speed_ms,0,blend_radius_m)
    |   movel([0.304245, -1.288646, -2.631026, -0.792717, 1.570796, 1.875042],accel_mss,speed_ms,0,blend_radius_m)
    |   movel([0.303498, -1.289482, -2.630540, -0.792367, 1.570796, 1.874294],accel_mss,speed_ms,0,blend_radius_m)
    |   movel([0.297361, -1.295291, -2.627137, -0.789960, 1.570796, 1.868158],accel_mss,speed_ms,0,blend_radius_m)
    |   movel([0.295022, -1.297584, -2.625783, -0.789022, 1.570796, 1.865818],accel_mss,speed_ms,0,blend_radius_m)
    |   movel([0.293022, -1.299671, -2.624544, -0.788174, 1.570796, 1.863818],accel_mss,speed_ms,0,blend_radius_m)
    |   movel([0.294092, -1.298834, -2.625041, -0.788514, 1.570796, 1.864888],accel_mss,speed_ms,0,blend_radius_m)
    |   movel([0.300252, -1.294127, -2.627823, -0.790439, 1.570796, 1.871048],accel_mss,speed_ms,0,blend_radius_m)
    |   movel([0.302053, -1.292828, -2.628585, -0.790976, 1.570796, 1.872849],accel_mss,speed_ms,0,blend_radius_m)
    |   movel([0.306675, -1.289633, -2.630452, -0.792304, 1.570796, 1.877471],accel_mss,speed_ms,0,blend_radius_m)
    |   movel([0.307641, -1.289074, -2.630777, -0.792538, 1.570796, 1.878437],accel_mss,speed_ms,0,blend_radius_m)
    |   movel([0.308002, -1.289066, -2.630781, -0.792541, 1.570796, 1.878799],accel_mss,speed_ms,0,blend_radius_m)
    |   movel([0.308075, -1.289156, -2.630729, -0.792504, 1.570796, 1.878872],accel_mss,speed_ms,0,blend_radius_m)
    |   movel([0.308126, -1.289495, -2.630532, -0.792362, 1.570796, 1.878922],accel_mss,speed_ms,0,blend_radius_m)
    |   movel([0.308008, -1.289654, -2.630439, -0.792295, 1.570796, 1.878804],accel_mss,speed_ms,0,blend_radius_m)
    |   movel([0.304596, -1.292114, -2.629003, -0.791271, 1.570796, 1.875393],accel_mss,speed_ms,0,blend_radius_m)
    |   movel([0.301963, -1.293982, -2.627908, -0.790499, 1.570796, 1.872759],accel_mss,speed_ms,0,blend_radius_m)
    |   speed_ms = 0.005
    |   movel([0.301963, -1.284735, -2.623521, -0.804133, 1.570796, 1.872759],accel_mss,speed_ms,0,blend_radius_m)
    |   speed_ms = 0.040
    |   movel([0.304558, -1.293744, -2.618245, -0.800400, 1.570796, 1.875354],accel_mss,speed_ms,0,blend_radius_m)
    |   speed_ms = 0.005
    |   movel([0.304558, -1.302941, -2.622591, -0.786857, 1.570796, 1.875354],accel_mss,speed_ms,0,blend_radius_m)
    |   speed_ms = 0.025
    |   movel([0.305417, -1.302454, -2.622883, -0.787052, 1.570796, 1.876213],accel_mss,speed_ms,0,blend_radius_m)
    |   movel([0.306402, -1.301783, -2.623284, -0.787322, 1.570796, 1.877198],accel_mss,speed_ms,0,blend_radius_m)
    |   movel([0.306548, -1.301581, -2.623405, -0.787403, 1.570796, 1.877344],accel_mss,speed_ms,0,blend_radius_m)
    |   movel([0.306544, -1.301369, -2.623532, -0.787488, 1.570796, 1.877340],accel_mss,speed_ms,0,blend_radius_m)
    |   movel([0.306386, -1.301266, -2.623593, -0.787530, 1.570796, 1.877182],accel_mss,speed_ms,0,blend_radius_m)
    |   movel([0.305731, -1.301370, -2.623531, -0.787488, 1.570796, 1.876527],accel_mss,speed_ms,0,blend_radius_m)
    |   movel([0.304347, -1.302044, -2.623128, -0.787217, 1.570796, 1.875144],accel_mss,speed_ms,0,blend_radius_m)
    |   movel([0.299921, -1.304729, -2.621518, -0.786143, 1.570796, 1.870718],accel_mss,speed_ms,0,blend_radius_m)
    |   movel([0.297564, -1.306321, -2.620559, -0.785510, 1.570796, 1.868360],accel_mss,speed_ms,0,blend_radius_m)
    |   movel([0.287265, -1.313737, -2.616045, -0.782607, 1.570796, 1.858062],accel_mss,speed_ms,0,blend_radius_m)
    |   movel([0.287278, -1.313501, -2.616190, -0.782698, 1.570796, 1.858075],accel_mss,speed_ms,0,blend_radius_m)
    |   movel([0.291163, -1.309758, -2.618476, -0.784155, 1.570796, 1.861959],accel_mss,speed_ms,0,blend_radius_m)
    |   movel([0.299271, -1.302210, -2.623029, -0.787150, 1.570796, 1.870067],accel_mss,speed_ms,0,blend_radius_m)
    |   movel([0.299999, -1.301506, -2.623450, -0.787433, 1.570796, 1.870795],accel_mss,speed_ms,0,blend_radius_m)
    |   movel([0.300715, -1.300697, -2.623933, -0.787759, 1.570796, 1.871512],accel_mss,speed_ms,0,blend_radius_m)
    |   movel([0.300814, -1.300531, -2.624032, -0.787826, 1.570796, 1.871610],accel_mss,speed_ms,0,blend_radius_m)
    |   movel([0.301697, -1.299852, -2.624436, -0.788101, 1.570796, 1.872493],accel_mss,speed_ms,0,blend_radius_m)
    |   movel([0.302356, -1.299433, -2.624686, -0.788271, 1.570796, 1.873152],accel_mss,speed_ms,0,blend_radius_m)
    |   movel([0.302701, -1.299113, -2.624876, -0.788400, 1.570796, 1.873497],accel_mss,speed_ms,0,blend_radius_m)
    |   movel([0.302809, -1.298840, -2.625038, -0.788511, 1.570796, 1.873605],accel_mss,speed_ms,0,blend_radius_m)
    |   movel([0.302563, -1.298472, -2.625256, -0.788661, 1.570796, 1.873359],accel_mss,speed_ms,0,blend_radius_m)
    |   movel([0.302381, -1.298474, -2.625255, -0.788660, 1.570796, 1.873177],accel_mss,speed_ms,0,blend_radius_m)
    |   movel([0.301476, -1.298956, -2.624969, -0.788464, 1.570796, 1.872272],accel_mss,speed_ms,0,blend_radius_m)
    |   movel([0.300007, -1.299882, -2.624418, -0.788089, 1.570796, 1.870803],accel_mss,speed_ms,0,blend_radius_m)
    |   movel([0.296100, -1.302572, -2.622812, -0.787005, 1.570796, 1.866896],accel_mss,speed_ms,0,blend_radius_m)
    |   movel([0.294444, -1.303797, -2.622078, -0.786514, 1.570796, 1.865240],accel_mss,speed_ms,0,blend_radius_m)
    |   movel([0.292521, -1.305229, -2.621216, -0.785943, 1.570796, 1.863317],accel_mss,speed_ms,0,blend_radius_m)
    |   movel([0.297537, -1.299514, -2.624637, -0.788238, 1.570796, 1.868333],accel_mss,speed_ms,0,blend_radius_m)
    |   movel([0.298252, -1.298745, -2.625094, -0.788550, 1.570796, 1.869048],accel_mss,speed_ms,0,blend_radius_m)
    |   movel([0.300320, -1.296702, -2.626305, -0.789382, 1.570796, 1.871116],accel_mss,speed_ms,0,blend_radius_m)
    |   movel([0.301058, -1.296007, -2.626715, -0.789667, 1.570796, 1.871854],accel_mss,speed_ms,0,blend_radius_m)
    |   movel([0.301392, -1.295531, -2.626996, -0.789862, 1.570796, 1.872188],accel_mss,speed_ms,0,blend_radius_m)
    |   movel([0.301351, -1.295278, -2.627145, -0.789966, 1.570796, 1.872147],accel_mss,speed_ms,0,blend_radius_m)
    |   movel([0.300993, -1.295225, -2.627177, -0.789988, 1.570796, 1.871789],accel_mss,speed_ms,0,blend_radius_m)
    |   movel([0.300409, -1.295491, -2.627020, -0.789878, 1.570796, 1.871205],accel_mss,speed_ms,0,blend_radius_m)
    |   movel([0.299464, -1.296294, -2.626546, -0.789549, 1.570796, 1.870261],accel_mss,speed_ms,0,blend_radius_m)
    |   movel([0.298172, -1.297576, -2.625787, -0.789025, 1.570796, 1.868968],accel_mss,speed_ms,0,blend_radius_m)
    |   movel([0.292606, -1.303730, -2.622118, -0.786541, 1.570796, 1.863402],accel_mss,speed_ms,0,blend_radius_m)
    |   movel([0.290489, -1.306225, -2.620616, -0.785548, 1.570796, 1.861285],accel_mss,speed_ms,0,blend_radius_m)
    |   movel([0.289248, -1.307852, -2.619633, -0.784905, 1.570796, 1.860044],accel_mss,speed_ms,0,blend_radius_m)
    |   movel([0.289051, -1.308229, -2.619404, -0.784756, 1.570796, 1.859847],accel_mss,speed_ms,0,blend_radius_m)
    |   movel([0.289003, -1.308586, -2.619188, -0.784615, 1.570796, 1.859800],accel_mss,speed_ms,0,blend_radius_m)
    |   movel([0.289200, -1.308759, -2.619083, -0.784548, 1.570796, 1.859997],accel_mss,speed_ms,0,blend_radius_m)
    |   movel([0.289614, -1.308636, -2.619157, -0.784596, 1.570796, 1.860410],accel_mss,speed_ms,0,blend_radius_m)
    |   movel([0.290420, -1.308087, -2.619490, -0.784812, 1.570796, 1.861217],accel_mss,speed_ms,0,blend_radius_m)
    |   movel([0.293727, -1.305444, -2.621087, -0.785858, 1.570796, 1.864523],accel_mss,speed_ms,0,blend_radius_m)
    |   movel([0.295240, -1.304265, -2.621797, -0.786328, 1.570796, 1.866037],accel_mss,speed_ms,0,blend_radius_m)
    |   movel([0.297126, -1.302893, -2.622620, -0.786876, 1.570796, 1.867923],accel_mss,speed_ms,0,blend_radius_m)
    |   movel([0.295161, -1.304789, -2.621481, -0.786118, 1.570796, 1.865957],accel_mss,speed_ms,0,blend_radius_m)
    |   movel([0.291291, -1.308444, -2.619274, -0.784671, 1.570796, 1.862088],accel_mss,speed_ms,0,blend_radius_m)
    |   movel([0.286988, -1.312718, -2.616670, -0.783001, 1.570796, 1.857784],accel_mss,speed_ms,0,blend_radius_m)
    |   movel([0.282863, -1.316935, -2.614077, -0.781377, 1.570796, 1.853659],accel_mss,speed_ms,0,blend_radius_m)
    |   movel([0.282544, -1.317340, -2.613827, -0.781222, 1.570796, 1.853340],accel_mss,speed_ms,0,blend_radius_m)
    |   movel([0.282347, -1.317767, -2.613563, -0.781059, 1.570796, 1.853143],accel_mss,speed_ms,0,blend_radius_m)
    |   movel([0.282361, -1.317934, -2.613460, -0.780996, 1.570796, 1.853157],accel_mss,speed_ms,0,blend_radius_m)
    |   movel([0.282506, -1.317997, -2.613420, -0.780972, 1.570796, 1.853302],accel_mss,speed_ms,0,blend_radius_m)
    |   movel([0.283054, -1.317835, -2.613521, -0.781034, 1.570796, 1.853850],accel_mss,speed_ms,0,blend_radius_m)
    |   movel([0.284251, -1.317070, -2.613993, -0.781325, 1.570796, 1.855047],accel_mss,speed_ms,0,blend_radius_m)
    |   movel([0.286428, -1.315474, -2.614978, -0.781937, 1.570796, 1.857224],accel_mss,speed_ms,0,blend_radius_m)
    |   movel([0.290679, -1.312301, -2.616925, -0.783163, 1.570796, 1.861475],accel_mss,speed_ms,0,blend_radius_m)
    |   movel([0.291209, -1.311954, -2.617137, -0.783298, 1.570796, 1.862005],accel_mss,speed_ms,0,blend_radius_m)
    |   movel([0.285869, -1.317658, -2.613630, -0.781101, 1.570796, 1.856665],accel_mss,speed_ms,0,blend_radius_m)
    |   movel([0.284109, -1.319646, -2.612397, -0.780345, 1.570796, 1.854906],accel_mss,speed_ms,0,blend_radius_m)
    |   movel([0.280897, -1.323503, -2.609992, -0.778894, 1.570796, 1.851693],accel_mss,speed_ms,0,blend_radius_m)
    |   movel([0.280283, -1.324365, -2.609451, -0.778573, 1.570796, 1.851079],accel_mss,speed_ms,0,blend_radius_m)
    |   movel([0.280101, -1.324830, -2.609159, -0.778400, 1.570796, 1.850897],accel_mss,speed_ms,0,blend_radius_m)
    |   movel([0.280243, -1.325060, -2.609015, -0.778314, 1.570796, 1.851040],accel_mss,speed_ms,0,blend_radius_m)
    |   movel([0.280547, -1.324993, -2.609057, -0.778339, 1.570796, 1.851343],accel_mss,speed_ms,0,blend_radius_m)
    |   movel([0.281120, -1.324605, -2.609300, -0.778483, 1.570796, 1.851917],accel_mss,speed_ms,0,blend_radius_m)
    |   movel([0.285734, -1.320954, -2.611584, -0.779851, 1.570796, 1.856531],accel_mss,speed_ms,0,blend_radius_m)
    |   movel([0.290005, -1.317612, -2.613659, -0.781119, 1.570796, 1.860802],accel_mss,speed_ms,0,blend_radius_m)
    |   movel([0.297334, -1.312251, -2.616955, -0.783182, 1.570796, 1.868130],accel_mss,speed_ms,0,blend_radius_m)
    |   movel([0.298736, -1.311482, -2.617425, -0.783482, 1.570796, 1.869532],accel_mss,speed_ms,0,blend_radius_m)
    |   movel([0.299041, -1.311258, -2.617562, -0.783569, 1.570796, 1.869838],accel_mss,speed_ms,0,blend_radius_m)
    |   movel([0.299206, -1.310939, -2.617757, -0.783694, 1.570796, 1.870002],accel_mss,speed_ms,0,blend_radius_m)
    |   movel([0.299157, -1.310661, -2.617926, -0.783802, 1.570796, 1.869954],accel_mss,speed_ms,0,blend_radius_m)
    |   movel([0.298913, -1.310558, -2.617989, -0.783842, 1.570796, 1.869709],accel_mss,speed_ms,0,blend_radius_m)
    |   movel([0.298423, -1.310647, -2.617935, -0.783807, 1.570796, 1.869219],accel_mss,speed_ms,0,blend_radius_m)
    |   movel([0.297918, -1.310892, -2.617785, -0.783712, 1.570796, 1.868714],accel_mss,speed_ms,0,blend_radius_m)
    |   movel([0.295201, -1.312723, -2.616667, -0.782999, 1.570796, 1.865998],accel_mss,speed_ms,0,blend_radius_m)
    |   movel([0.291601, -1.315336, -2.615063, -0.781990, 1.570796, 1.862397],accel_mss,speed_ms,0,blend_radius_m)
    |   movel([0.286866, -1.318973, -2.612815, -0.780600, 1.570796, 1.857662],accel_mss,speed_ms,0,blend_radius_m)
    |   movel([0.284311, -1.320966, -2.611577, -0.779847, 1.570796, 1.855107],accel_mss,speed_ms,0,blend_radius_m)
    |   movel([0.284177, -1.320950, -2.611586, -0.779852, 1.570796, 1.854973],accel_mss,speed_ms,0,blend_radius_m)
    |   movel([0.284275, -1.320718, -2.611731, -0.779940, 1.570796, 1.855071],accel_mss,speed_ms,0,blend_radius_m)
    |   movel([0.286791, -1.317929, -2.613462, -0.780997, 1.570796, 1.857587],accel_mss,speed_ms,0,blend_radius_m)
    |   movel([0.288241, -1.316349, -2.614439, -0.781601, 1.570796, 1.859038],accel_mss,speed_ms,0,blend_radius_m)
    |   movel([0.293255, -1.311292, -2.617541, -0.783556, 1.570796, 1.864051],accel_mss,speed_ms,0,blend_radius_m)
    |   movel([0.293701, -1.310801, -2.617841, -0.783747, 1.570796, 1.864497],accel_mss,speed_ms,0,blend_radius_m)
    |   movel([0.294034, -1.310210, -2.618201, -0.783978, 1.570796, 1.864830],accel_mss,speed_ms,0,blend_radius_m)
    |   movel([0.294135, -1.309959, -2.618353, -0.784077, 1.570796, 1.864931],accel_mss,speed_ms,0,blend_radius_m)
    |   movel([0.294465, -1.309624, -2.618557, -0.784208, 1.570796, 1.865262],accel_mss,speed_ms,0,blend_radius_m)
    |   movel([0.295090, -1.309125, -2.618861, -0.784404, 1.570796, 1.865886],accel_mss,speed_ms,0,blend_radius_m)
    |   movel([0.298565, -1.306673, -2.620346, -0.785370, 1.570796, 1.869361],accel_mss,speed_ms,0,blend_radius_m)
    |   movel([0.300735, -1.305237, -2.621212, -0.785940, 1.570796, 1.871532],accel_mss,speed_ms,0,blend_radius_m)
    |   movel([0.304558, -1.302941, -2.622591, -0.786857, 1.570796, 1.875354],accel_mss,speed_ms,0,blend_radius_m)
    |   movel([0.305417, -1.302454, -2.622883, -0.787052, 1.570796, 1.876213],accel_mss,speed_ms,0,blend_radius_m)
    |   movel([0.306402, -1.301783, -2.623284, -0.787322, 1.570796, 1.877198],accel_mss,speed_ms,0,blend_radius_m)
    |   movel([0.306548, -1.301581, -2.623405, -0.787403, 1.570796, 1.877344],accel_mss,speed_ms,0,blend_radius_m)
    |   movel([0.306544, -1.301369, -2.623532, -0.787488, 1.570796, 1.877340],accel_mss,speed_ms,0,blend_radius_m)
    |   movel([0.306386, -1.301266, -2.623593, -0.787530, 1.570796, 1.877182],accel_mss,speed_ms,0,blend_radius_m)
    |   speed_ms = 0.005
    |   movel([0.306386, -1.292060, -2.619239, -0.801090, 1.570796, 1.877182],accel_mss,speed_ms,0,blend_radius_m)
    |   speed_ms = 0.040
    |   movel([0.303574, -1.299558, -2.614785, -0.798045, 1.570796, 1.874370],accel_mss,speed_ms,0,blend_radius_m)
    |   speed_ms = 0.005
    |   movel([0.303574, -1.308721, -2.619106, -0.784562, 1.570796, 1.874370],accel_mss,speed_ms,0,blend_radius_m)
    |   speed_ms = 0.025
    |   movel([0.304542, -1.307814, -2.619655, -0.784919, 1.570796, 1.875338],accel_mss,speed_ms,0,blend_radius_m)
    |   movel([0.305048, -1.307189, -2.620034, -0.785166, 1.570796, 1.875844],accel_mss,speed_ms,0,blend_radius_m)
    |   movel([0.305096, -1.306861, -2.620232, -0.785296, 1.570796, 1.875893],accel_mss,speed_ms,0,blend_radius_m)
    |   movel([0.304816, -1.306752, -2.620298, -0.785339, 1.570796, 1.875613],accel_mss,speed_ms,0,blend_radius_m)
    |   movel([0.304512, -1.306872, -2.620226, -0.785292, 1.570796, 1.875308],accel_mss,speed_ms,0,blend_radius_m)
    |   movel([0.304017, -1.307227, -2.620011, -0.785151, 1.570796, 1.874813],accel_mss,speed_ms,0,blend_radius_m)
    |   movel([0.303333, -1.307795, -2.619667, -0.784927, 1.570796, 1.874129],accel_mss,speed_ms,0,blend_radius_m)
    |   movel([0.298799, -1.312087, -2.617056, -0.783246, 1.570796, 1.869596],accel_mss,speed_ms,0,blend_radius_m)
    |   movel([0.295219, -1.315804, -2.614775, -0.781810, 1.570796, 1.866015],accel_mss,speed_ms,0,blend_radius_m)
    |   movel([0.291562, -1.319882, -2.612251, -0.780256, 1.570796, 1.862358],accel_mss,speed_ms,0,blend_radius_m)
    |   movel([0.287774, -1.324381, -2.609441, -0.778567, 1.570796, 1.858570],accel_mss,speed_ms,0,blend_radius_m)
    |   movel([0.284773, -1.327994, -2.607165, -0.777230, 1.570796, 1.855570],accel_mss,speed_ms,0,blend_radius_m)
    |   movel([0.284826, -1.327831, -2.607268, -0.777290, 1.570796, 1.855622],accel_mss,speed_ms,0,blend_radius_m)
    |   movel([0.285459, -1.326761, -2.607944, -0.777684, 1.570796, 1.856255],accel_mss,speed_ms,0,blend_radius_m)
    |   movel([0.289831, -1.319966, -2.612199, -0.780224, 1.570796, 1.860627],accel_mss,speed_ms,0,blend_radius_m)
    |   movel([0.290053, -1.319481, -2.612500, -0.780408, 1.570796, 1.860850],accel_mss,speed_ms,0,blend_radius_m)
    |   movel([0.289996, -1.319251, -2.612643, -0.780495, 1.570796, 1.860792],accel_mss,speed_ms,0,blend_radius_m)
    |   movel([0.289703, -1.319199, -2.612675, -0.780515, 1.570796, 1.860499],accel_mss,speed_ms,0,blend_radius_m)
    |   movel([0.289241, -1.319466, -2.612509, -0.780413, 1.570796, 1.860037],accel_mss,speed_ms,0,blend_radius_m)
    |   movel([0.288528, -1.320353, -2.611958, -0.780078, 1.570796, 1.859324],accel_mss,speed_ms,0,blend_radius_m)
    |   movel([0.287484, -1.321879, -2.611007, -0.779503, 1.570796, 1.858281],accel_mss,speed_ms,0,blend_radius_m)
    |   movel([0.285710, -1.324682, -2.609252, -0.778455, 1.570796, 1.856506],accel_mss,speed_ms,0,blend_radius_m)
    |   movel([0.282417, -1.330281, -2.605715, -0.776393, 1.570796, 1.853214],accel_mss,speed_ms,0,blend_radius_m)
    |   movel([0.281248, -1.332490, -2.604308, -0.775591, 1.570796, 1.852044],accel_mss,speed_ms,0,blend_radius_m)
    |   movel([0.281185, -1.333010, -2.603976, -0.775403, 1.570796, 1.851981],accel_mss,speed_ms,0,blend_radius_m)
    |   movel([0.281242, -1.333104, -2.603916, -0.775369, 1.570796, 1.852038],accel_mss,speed_ms,0,blend_radius_m)
    |   movel([0.281542, -1.333227, -2.603837, -0.775325, 1.570796, 1.852338],accel_mss,speed_ms,0,blend_radius_m)
    |   movel([0.281717, -1.333125, -2.603902, -0.775362, 1.570796, 1.852513],accel_mss,speed_ms,0,blend_radius_m)
    |   movel([0.285200, -1.328931, -2.606572, -0.776886, 1.570796, 1.855996],accel_mss,speed_ms,0,blend_radius_m)
    |   movel([0.290563, -1.322384, -2.610692, -0.779313, 1.570796, 1.861359],accel_mss,speed_ms,0,blend_radius_m)
    |   movel([0.295241, -1.317031, -2.614017, -0.781340, 1.570796, 1.866037],accel_mss,speed_ms,0,blend_radius_m)
    |   movel([0.299498, -1.312559, -2.616767, -0.783063, 1.570796, 1.870295],accel_mss,speed_ms,0,blend_radius_m)
    |   movel([0.303574, -1.308721, -2.619106, -0.784562, 1.570796, 1.874370],accel_mss,speed_ms,0,blend_radius_m)
    |   movel([0.304542, -1.307814, -2.619655, -0.784919, 1.570796, 1.875338],accel_mss,speed_ms,0,blend_radius_m)
    |   movel([0.305048, -1.307189, -2.620034, -0.785166, 1.570796, 1.875844],accel_mss,speed_ms,0,blend_radius_m)
    |   movel([0.305096, -1.306861, -2.620232, -0.785296, 1.570796, 1.875893],accel_mss,speed_ms,0,blend_radius_m)
    |   movel([0.304816, -1.306752, -2.620298, -0.785339, 1.570796, 1.875613],accel_mss,speed_ms,0,blend_radius_m)
    |   speed_ms = 0.005
    |   movel([0.304816, -1.297577, -2.615969, -0.798843, 1.570796, 1.875613],accel_mss,speed_ms,0,blend_radius_m)
    |   speed_ms = 0.040
    |   movel([0.299752, -1.309796, -2.608588, -0.794005, 1.570796, 1.870548],accel_mss,speed_ms,0,blend_radius_m)
    |   speed_ms = 0.005
    |   movel([0.299752, -1.318898, -2.612862, -0.780629, 1.570796, 1.870548],accel_mss,speed_ms,0,blend_radius_m)
    |   speed_ms = 0.025
    |   movel([0.296568, -1.321749, -2.611088, -0.779552, 1.570796, 1.867364],accel_mss,speed_ms,0,blend_radius_m)
    |   movel([0.293386, -1.324901, -2.609115, -0.778373, 1.570796, 1.864183],accel_mss,speed_ms,0,blend_radius_m)
    |   movel([0.290009, -1.328555, -2.606810, -0.777024, 1.570796, 1.860805],accel_mss,speed_ms,0,blend_radius_m)
    |   movel([0.286235, -1.332925, -2.604030, -0.775434, 1.570796, 1.857032],accel_mss,speed_ms,0,blend_radius_m)
    |   movel([0.283751, -1.335746, -2.602222, -0.774421, 1.570796, 1.854548],accel_mss,speed_ms,0,blend_radius_m)
    |   movel([0.283601, -1.335830, -2.602168, -0.774391, 1.570796, 1.854398],accel_mss,speed_ms,0,blend_radius_m)
    |   movel([0.283307, -1.335740, -2.602226, -0.774423, 1.570796, 1.854104],accel_mss,speed_ms,0,blend_radius_m)
    |   movel([0.283261, -1.335423, -2.602430, -0.774537, 1.570796, 1.854057],accel_mss,speed_ms,0,blend_radius_m)
    |   movel([0.283525, -1.334743, -2.602866, -0.774780, 1.570796, 1.854321],accel_mss,speed_ms,0,blend_radius_m)
    |   movel([0.284237, -1.333401, -2.603726, -0.775262, 1.570796, 1.855033],accel_mss,speed_ms,0,blend_radius_m)
    |   movel([0.286300, -1.329291, -2.606344, -0.776754, 1.570796, 1.857097],accel_mss,speed_ms,0,blend_radius_m)
    |   movel([0.287406, -1.326866, -2.607877, -0.777645, 1.570796, 1.858202],accel_mss,speed_ms,0,blend_radius_m)
    |   movel([0.287762, -1.326183, -2.608308, -0.777898, 1.570796, 1.858559],accel_mss,speed_ms,0,blend_radius_m)
    |   movel([0.288040, -1.325875, -2.608502, -0.778012, 1.570796, 1.858836],accel_mss,speed_ms,0,blend_radius_m)
    |   movel([0.288385, -1.325722, -2.608598, -0.778069, 1.570796, 1.859181],accel_mss,speed_ms,0,blend_radius_m)
    |   movel([0.288639, -1.325714, -2.608603, -0.778072, 1.570796, 1.859435],accel_mss,speed_ms,0,blend_radius_m)
    |   movel([0.288719, -1.325971, -2.608442, -0.777977, 1.570796, 1.859515],accel_mss,speed_ms,0,blend_radius_m)
    |   movel([0.288549, -1.326456, -2.608136, -0.777797, 1.570796, 1.859345],accel_mss,speed_ms,0,blend_radius_m)
    |   movel([0.286617, -1.330953, -2.605288, -0.776148, 1.570796, 1.857414],accel_mss,speed_ms,0,blend_radius_m)
    |   movel([0.286887, -1.330800, -2.605385, -0.776204, 1.570796, 1.857684],accel_mss,speed_ms,0,blend_radius_m)
    |   movel([0.287150, -1.330523, -2.605562, -0.776305, 1.570796, 1.857946],accel_mss,speed_ms,0,blend_radius_m)
    |   movel([0.291273, -1.325921, -2.608473, -0.777995, 1.570796, 1.862069],accel_mss,speed_ms,0,blend_radius_m)
    |   movel([0.293502, -1.323565, -2.609953, -0.778871, 1.570796, 1.864299],accel_mss,speed_ms,0,blend_radius_m)
    |   movel([0.296875, -1.320310, -2.611985, -0.780094, 1.570796, 1.867671],accel_mss,speed_ms,0,blend_radius_m)
    |   movel([0.299030, -1.318418, -2.613160, -0.780812, 1.570796, 1.869826],accel_mss,speed_ms,0,blend_radius_m)
    |   movel([0.301124, -1.316640, -2.614259, -0.781490, 1.570796, 1.871920],accel_mss,speed_ms,0,blend_radius_m)
    |   movel([0.301941, -1.316067, -2.614613, -0.781710, 1.570796, 1.872737],accel_mss,speed_ms,0,blend_radius_m)
    |   movel([0.302201, -1.315983, -2.614664, -0.781741, 1.570796, 1.872997],accel_mss,speed_ms,0,blend_radius_m)
    |   movel([0.302461, -1.316022, -2.614640, -0.781727, 1.570796, 1.873258],accel_mss,speed_ms,0,blend_radius_m)
    |   movel([0.302636, -1.316157, -2.614557, -0.781675, 1.570796, 1.873433],accel_mss,speed_ms,0,blend_radius_m)
    |   movel([0.302654, -1.316348, -2.614439, -0.781602, 1.570796, 1.873450],accel_mss,speed_ms,0,blend_radius_m)
    |   movel([0.301782, -1.317151, -2.613944, -0.781295, 1.570796, 1.872579],accel_mss,speed_ms,0,blend_radius_m)
    |   movel([0.300850, -1.317961, -2.613443, -0.780985, 1.570796, 1.871646],accel_mss,speed_ms,0,blend_radius_m)
    |   movel([0.299752, -1.318898, -2.612862, -0.780629, 1.570796, 1.870548],accel_mss,speed_ms,0,blend_radius_m)
    |   movel([0.297425, -1.320980, -2.611568, -0.779841, 1.570796, 1.868221],accel_mss,speed_ms,0,blend_radius_m)
    |   speed_ms = 0.005
    |   movel([0.297425, -1.311891, -2.607303, -0.793196, 1.570796, 1.868221],accel_mss,speed_ms,0,blend_radius_m)
    |   speed_ms = 0.040
    |   movel([0.326144, -1.292156, -2.619183, -0.801050, 1.570796, 1.896941],accel_mss,speed_ms,0,blend_radius_m)
    |   speed_ms = 0.005
    |   movel([0.326144, -1.301362, -2.623536, -0.787491, 1.570796, 1.896941],accel_mss,speed_ms,0,blend_radius_m)
    |   speed_ms = 0.025
    |   movel([0.325589, -1.301882, -2.623225, -0.787282, 1.570796, 1.896385],accel_mss,speed_ms,0,blend_radius_m)
    |   movel([0.325038, -1.302447, -2.622887, -0.787055, 1.570796, 1.895835],accel_mss,speed_ms,0,blend_radius_m)
    |   movel([0.322806, -1.304745, -2.621508, -0.786136, 1.570796, 1.893602],accel_mss,speed_ms,0,blend_radius_m)
    |   movel([0.321385, -1.306021, -2.620739, -0.785629, 1.570796, 1.892181],accel_mss,speed_ms,0,blend_radius_m)
    |   movel([0.319735, -1.307298, -2.619968, -0.785123, 1.570796, 1.890531],accel_mss,speed_ms,0,blend_radius_m)
    |   movel([0.317347, -1.308974, -2.618952, -0.784463, 1.570796, 1.888143],accel_mss,speed_ms,0,blend_radius_m)
    |   movel([0.312713, -1.312267, -2.616946, -0.783176, 1.570796, 1.883510],accel_mss,speed_ms,0,blend_radius_m)
    |   movel([0.311397, -1.313348, -2.616284, -0.782757, 1.570796, 1.882194],accel_mss,speed_ms,0,blend_radius_m)
    |   movel([0.310253, -1.314435, -2.615617, -0.782337, 1.570796, 1.881049],accel_mss,speed_ms,0,blend_radius_m)
    |   movel([0.309323, -1.315477, -2.614976, -0.781936, 1.570796, 1.880120],accel_mss,speed_ms,0,blend_radius_m)
    |   movel([0.307590, -1.317877, -2.613495, -0.781018, 1.570796, 1.878386],accel_mss,speed_ms,0,blend_radius_m)
